(*

short summary
==================
This class tests all methods of REAL assertions
with various combinations of inputs and checks expected 
outputs are satisfied or not

.. <legal notes>

legal notes
=================
| SPDX-FileCopyrightText: © 2022 ekvip automation GmbH <info@ekvip.de>
| SPDX-License-Identifier: Apache-2.0
| For details check: Apache-2.0_

.. _Apache-2.0: https://www.apache.org/licenses/LICENSE-2.0

.. </legal notes>

methods and properties
======================

*)


FUNCTION_BLOCK RealAssertionTests EXTENDS AbstractAssertorTest
VAR
	(* not a number *)
	NAN							:REAL;
	(* infinity *)
	INF							:REAL;
	(* -infinity *)
	MINUS_INF					:REAL;
	(* -0.0 (MSB is set only) *)
	MINUS_ZERO					:REAL;
	(* minimum subnormal value (all fraction bits and MSB set only) *)
	MIN_SUBNORMAL				:REAL;
	(* maximum subnormal value (all fraction bits are set only) *)
	MAX_SUBNORMAL				:REAL;
	(* smallest positive subnormal value (LSB set only)*)
	SMALLEST_POSITIVE_SUBNORMAL	:REAL;
	(* smallest negative subnormal value (LSB and MSB set only)*)
	SMALLEST_NEGATIVE_SUBNORMAL	:REAL;
END_VAR
VAR CONSTANT
	(* prefix to unify the test names *)
	TEST_NAME_PREFIX					:STRING := 'assert.float.single.';
	(* max value of real *)
	MAX_NON_SPECIAL						:REAL := 3.402823E+38;
	(* min value of real *)
	MIN_NON_SPECIAL						:REAL := -3.402823E+38;
	(* 0.0 *)
	ZERO								:REAL := 0.0;
	(* 1% *)
	ONE_PERCENT							:REAL := 0.01;
	(* 1‰ *)
	ONE_PERMILLE						:REAL := 0.001;
	(* bit number of the sign bit *)
	SIGN								:USINT := 31;
	(* binary value of 0.0 *)
	BINARY_ZERO							:DWORD := 16#0000_0000;
	(* binary value of -0.0 *)
	BINARY_MINUS_ZERO					:DWORD := 16#8000_0000;
	(* binary value of inf *)
	BINARY_INFINITY						:DWORD := 16#7F80_0000;
	(* binary value of -inf *)
	BINARY_NEGATIVE_INFINITY			:DWORD := 16#FF80_0000;
	(* mask to filter the exponent of the number *)
	MASK_FOR_EXPONENT					:DWORD := 16#7F80_0000;
	(* minimum denormalized number *)
	BINARY_MIN_SUBNORMAL				:DWORD := 16#807F_FFFF;
	(* maximum denormalized number*)
	BINARY_MAX_SUBNORMAL				:DWORD := 16#007F_FFFF;
	(* smallest positive denormalizied number greater than zero *)
	BINARY_SMALLEST_POSITIVE_SUBNORMAL	:DWORD := 16#0000_0001;
	(* smallest negative denormalizied number greater than minus zero *)
	BINARY_SMALLEST_NEGATIVE_SUBNORMAL	:DWORD := 16#8000_0001;
	(* smallest positive signaling NaN *)
	BINARY_POSITIVE_SIGNALING_NAN		:DWORD := 16#7F80_0001;
END_VAR

THIS^.runValueIsEqualToTests();
THIS^.runValueIsGreaterThanTests();
THIS^.runValueIsInRangeOfTests();
THIS^.runValueIsLessThanTests();
THIS^.runValueIsMaxTests();
THIS^.runValueIsMinTests();
THIS^.runValueIsNotEqualToTests();
THIS^.runValueIsANumberTests();
THIS^.runValueIsFiniteTests();
THIS^.runValueIsInfiniteTests();
THIS^.runValueIsNaNTests();
THIS^.runValueIsNegativeTests();
THIS^.runValueIsPositiveTests();
THIS^.runValueIsNegativeInfiniteTests();
THIS^.runValueIsPositiveInfiniteTests();
THIS^.runValueIsNegativeZeroTests();
THIS^.runValueIsPositiveZeroTests();
THIS^.runValueIsNormalTests();
THIS^.runValueIsNotNegativeInfiniteTests();
THIS^.runValueIsNotPositiveInfiniteTests();
THIS^.runValueIsNotSpecialTests();
THIS^.runValueIsSpecialTests();
THIS^.runValueIsSubnormalTests();

(*

short summary
=============
It attaches the container with the class to test
and it sets the special numbers from `IEEE 754`_ standard

.. _IEEE 754: https://en.wikipedia.org/wiki/IEEE_754

legal notes
=================
| SPDX-FileCopyrightText: © 2023 ekvip automation GmbH <info@ekvip.de>
| SPDX-License-Identifier: Apache-2.0
| For details check: Apache-2.0_

.. _Apache-2.0: https://www.apache.org/licenses/LICENSE-2.0

.. </legal notes>

parameters
==========

*)

METHOD FB_init :BOOL
VAR_INPUT
	(* if TRUE, the retain variables are initialized (warm start / cold start) *)
    bInitRetains	:BOOL;
	(* if TRUE, the instance afterwards gets moved into the copy code (online change) *)
    bInCopyCode		:BOOL;
	(* container with the class to test *)
	classToBeTested :IAssertorContainer;
END_VAR
VAR
	{attribute 'hide'}
	newHashstate3		:CNM_AbstractObject.Hashcode;
	{attribute 'hide'}
	binaryNumberPointer	:POINTER TO DWORD;	
END_VAR
VAR CONSTANT
	{attribute 'hide'}
	NUMBER_OF_LEFT_SHIFTS		:UINT	:= 17;
	{attribute 'hide'}
	NUMBER_OF_LEFT_ROTATIONS	:UINT   := 45;
END_VAR
binaryNumberPointer := ADR(THIS^.NAN);
binaryNumberPointer^ := THIS^.BINARY_POSITIVE_SIGNALING_NAN;

binaryNumberPointer := ADR(THIS^.INF);
binaryNumberPointer^ := THIS^.BINARY_INFINITY;

binaryNumberPointer := ADR(THIS^.MINUS_INF);
binaryNumberPointer^ := THIS^.BINARY_NEGATIVE_INFINITY;

binaryNumberPointer := ADR(THIS^.MINUS_ZERO);
binaryNumberPointer^ := THIS^.BINARY_MINUS_ZERO;

binaryNumberPointer := ADR(THIS^.MIN_SUBNORMAL);
binaryNumberPointer^ := THIS^.BINARY_MIN_SUBNORMAL; 

binaryNumberPointer := ADR(THIS^.MAX_SUBNORMAL);
binaryNumberPointer^ := THIS^.BINARY_MAX_SUBNORMAL; 

binaryNumberPointer := ADR(THIS^.SMALLEST_POSITIVE_SUBNORMAL);
binaryNumberPointer^ := THIS^.BINARY_SMALLEST_POSITIVE_SUBNORMAL; 

binaryNumberPointer := ADR(THIS^.SMALLEST_NEGATIVE_SUBNORMAL);
binaryNumberPointer^ := THIS^.BINARY_SMALLEST_NEGATIVE_SUBNORMAL;
END_METHOD

(*

short summary
==================
This test method is a helper function to create a unified test name

.. <legal notes>

legal notes
=================
| SPDX-FileCopyrightText: © 2022 ekvip automation GmbH <info@ekvip.de>
| SPDX-License-Identifier: Apache-2.0
| For details check: Apache-2.0_

.. _Apache-2.0: https://www.apache.org/licenses/LICENSE-2.0

.. </legal notes>

parameters
==========

*)

METHOD PROTECTED getTestNameFor :Tc2_System.T_MaxString
VAR_INPUT
	(* name of the method to test, to create a unified test name *)
	nameOfMethodToTest	:Tc2_System.T_MaxString;
END_VAR
getTestNameFor := Tc2_Standard.CONCAT(THIS^.TEST_NAME_PREFIX, nameOfMethodToTest);
END_METHOD

(*

short summary
==================
This test method tests ``assert.float.single.valueIsANumber``
method of CNM_AssertionInterfaces library with various inputs

.. <legal notes>

legal notes
=================
| SPDX-FileCopyrightText: © 2022 ekvip automation GmbH <info@ekvip.de>
| SPDX-License-Identifier: Apache-2.0
| For details check: Apache-2.0_

.. _Apache-2.0: https://www.apache.org/licenses/LICENSE-2.0

.. </legal notes>

*)

METHOD runValueIsANumberTests
RETURN (NOT TcUnit.TEST_ORDERED(THIS^.getTestNameFor('valueIsANumber')));

THIS^.testValueIsANumber(THIS^.NAN);
THIS^.testValueIsANumber(THIS^.INF);
THIS^.testValueIsANumber(THIS^.MINUS_INF);
THIS^.testValueIsANumber(THIS^.MAX_NON_SPECIAL);
THIS^.testValueIsANumber(THIS^.MIN_NON_SPECIAL);
THIS^.testValueIsANumber(THIS^.ZERO);
THIS^.testValueIsANumber(THIS^.MINUS_ZERO);
THIS^.testValueIsANumber(THIS^.MAX_SUBNORMAL);
THIS^.testValueIsANumber(THIS^.MIN_SUBNORMAL);
THIS^.testValueIsANumber(THIS^.SMALLEST_NEGATIVE_SUBNORMAL);
THIS^.testValueIsANumber(THIS^.SMALLEST_POSITIVE_SUBNORMAL);
THIS^.testValueIsANumber(THIS^.ONE_PERCENT);
THIS^.testValueIsANumber(THIS^.ONE_PERMILLE);
THIS^.testValueIsANumber(THIS^.ONE_PERCENT * -1.0);
THIS^.testValueIsANumber(THIS^.ONE_PERMILLE * -1.0);

TcUnit.TEST_FINISHED();
END_METHOD

(*

short summary
==================
This test method tests ``assert.float.single.valueIsEqualTo``
method of CNM_AssertionInterfaces library with various inputs

.. <legal notes>

legal notes
=================
| SPDX-FileCopyrightText: © 2022 ekvip automation GmbH <info@ekvip.de>
| SPDX-License-Identifier: Apache-2.0
| For details check: Apache-2.0_

.. _Apache-2.0: https://www.apache.org/licenses/LICENSE-2.0

.. </legal notes>

*)

METHOD runValueIsEqualToTests
RETURN (NOT TcUnit.TEST_ORDERED(THIS^.getTestNameFor('valueIsEqualTo')));

THIS^.testValueIsEqualTo(
	valueToTest := THIS^.NAN,
	expected := THIS^.ONE_PERCENT,
	tolerance := THIS^.ONE_PERMILLE
);

THIS^.testValueIsEqualTo(
	valueToTest := THIS^.ONE_PERCENT,
	expected := THIS^.NAN,
	tolerance := THIS^.ONE_PERMILLE
);

THIS^.testValueIsEqualTo(
	valueToTest := THIS^.ONE_PERCENT,
	expected := THIS^.ONE_PERCENT,
	tolerance := THIS^.NAN
);

THIS^.testValueIsEqualTo(
	valueToTest := THIS^.NAN,
	expected := THIS^.NAN,
	tolerance := THIS^.ONE_PERCENT
);

THIS^.testValueIsEqualTo(
	valueToTest := THIS^.NAN,
	expected := THIS^.NAN,
	tolerance := THIS^.NAN
);

THIS^.testValueIsEqualTo(
	valueToTest := THIS^.INF,
	expected := THIS^.ONE_PERCENT,
	tolerance := THIS^.ONE_PERMILLE
);

THIS^.testValueIsEqualTo(
	valueToTest := THIS^.ONE_PERCENT,
	expected := THIS^.INF,
	tolerance := THIS^.ONE_PERMILLE
);

THIS^.testValueIsEqualTo(
	valueToTest := THIS^.ONE_PERCENT,
	expected := THIS^.ONE_PERCENT,
	tolerance := THIS^.INF
);

THIS^.testValueIsEqualTo(
	valueToTest := THIS^.INF,
	expected := THIS^.INF,
	tolerance := THIS^.ONE_PERCENT
);

THIS^.testValueIsEqualTo(
	valueToTest := THIS^.INF,
	expected := THIS^.INF,
	tolerance := THIS^.INF
);

THIS^.testValueIsEqualTo(
	valueToTest := THIS^.INF,
	expected := THIS^.MINUS_INF,
	tolerance := THIS^.INF
);

THIS^.testValueIsEqualTo(
	valueToTest := THIS^.MINUS_INF,
	expected := THIS^.ONE_PERCENT,
	tolerance := THIS^.ONE_PERMILLE
);

THIS^.testValueIsEqualTo(
	valueToTest := THIS^.ONE_PERCENT,
	expected := THIS^.MINUS_INF,
	tolerance := THIS^.ONE_PERMILLE
);

THIS^.testValueIsEqualTo(
	valueToTest := THIS^.ONE_PERCENT,
	expected := THIS^.ONE_PERCENT,
	tolerance := THIS^.MINUS_INF
);

THIS^.testValueIsEqualTo(
	valueToTest := THIS^.MINUS_INF,
	expected := THIS^.MINUS_INF,
	tolerance := THIS^.ONE_PERCENT
);

THIS^.testValueIsEqualTo(
	valueToTest := THIS^.MINUS_INF,
	expected := THIS^.MINUS_INF,
	tolerance := THIS^.MINUS_INF
);

THIS^.testValueIsEqualTo(
	valueToTest := THIS^.INF,
	expected := THIS^.MINUS_INF,
	tolerance := THIS^.INF
);

THIS^.testValueIsEqualTo(
	valueToTest := THIS^.MINUS_ZERO,
	expected := THIS^.SMALLEST_POSITIVE_SUBNORMAL,
	tolerance := THIS^.ONE_PERMILLE
);

THIS^.testValueIsEqualTo(
	valueToTest := THIS^.SMALLEST_POSITIVE_SUBNORMAL,
	expected := THIS^.MINUS_ZERO,
	tolerance := THIS^.ONE_PERMILLE
);

THIS^.testValueIsEqualTo(
	valueToTest := THIS^.SMALLEST_POSITIVE_SUBNORMAL,
	expected := THIS^.SMALLEST_POSITIVE_SUBNORMAL,
	tolerance := THIS^.MINUS_ZERO
);

THIS^.testValueIsEqualTo(
	valueToTest := THIS^.MINUS_ZERO,
	expected := THIS^.MINUS_ZERO,
	tolerance := THIS^.SMALLEST_POSITIVE_SUBNORMAL
);

THIS^.testValueIsEqualTo(
	valueToTest := THIS^.MINUS_ZERO,
	expected := THIS^.MINUS_ZERO,
	tolerance := THIS^.MINUS_ZERO
);

THIS^.testValueIsEqualTo(
	valueToTest := THIS^.MINUS_ZERO,
	expected := THIS^.ZERO,
	tolerance := THIS^.MINUS_ZERO
);

THIS^.testValueIsEqualTo(
	valueToTest := THIS^.ZERO,
	expected := THIS^.SMALLEST_POSITIVE_SUBNORMAL,
	tolerance := THIS^.ONE_PERMILLE
);

THIS^.testValueIsEqualTo(
	valueToTest := THIS^.SMALLEST_POSITIVE_SUBNORMAL,
	expected := THIS^.ZERO,
	tolerance := THIS^.ONE_PERMILLE
);

THIS^.testValueIsEqualTo(
	valueToTest := THIS^.SMALLEST_POSITIVE_SUBNORMAL,
	expected := THIS^.SMALLEST_POSITIVE_SUBNORMAL,
	tolerance := THIS^.ZERO
);

THIS^.testValueIsEqualTo(
	valueToTest := THIS^.ZERO,
	expected := THIS^.ZERO,
	tolerance := THIS^.SMALLEST_POSITIVE_SUBNORMAL
);

THIS^.testValueIsEqualTo(
	valueToTest := THIS^.ZERO,
	expected := THIS^.ZERO,
	tolerance := THIS^.ZERO
);

THIS^.testValueIsEqualTo(
	valueToTest := THIS^.ZERO,
	expected := THIS^.MINUS_ZERO,
	tolerance := THIS^.ZERO
);

THIS^.testValueIsEqualTo(
	valueToTest := THIS^.SMALLEST_POSITIVE_SUBNORMAL,
	expected := THIS^.ONE_PERCENT,
	tolerance := THIS^.ONE_PERMILLE
);

THIS^.testValueIsEqualTo(
	valueToTest := THIS^.ONE_PERCENT,
	expected := THIS^.SMALLEST_POSITIVE_SUBNORMAL,
	tolerance := THIS^.ONE_PERMILLE
);

THIS^.testValueIsEqualTo(
	valueToTest := THIS^.ONE_PERCENT,
	expected := THIS^.ONE_PERCENT,
	tolerance := THIS^.SMALLEST_POSITIVE_SUBNORMAL
);

THIS^.testValueIsEqualTo(
	valueToTest := THIS^.SMALLEST_POSITIVE_SUBNORMAL,
	expected := THIS^.SMALLEST_POSITIVE_SUBNORMAL,
	tolerance := THIS^.ONE_PERCENT
);

THIS^.testValueIsEqualTo(
	valueToTest := THIS^.SMALLEST_POSITIVE_SUBNORMAL,
	expected := THIS^.SMALLEST_POSITIVE_SUBNORMAL,
	tolerance := THIS^.SMALLEST_POSITIVE_SUBNORMAL
);

THIS^.testValueIsEqualTo(
	valueToTest := THIS^.SMALLEST_POSITIVE_SUBNORMAL,
	expected := THIS^.SMALLEST_NEGATIVE_SUBNORMAL,
	tolerance := THIS^.SMALLEST_POSITIVE_SUBNORMAL
);

THIS^.testValueIsEqualTo(
	valueToTest := THIS^.SMALLEST_NEGATIVE_SUBNORMAL,
	expected := THIS^.ONE_PERCENT,
	tolerance := THIS^.ONE_PERMILLE
);

THIS^.testValueIsEqualTo(
	valueToTest := THIS^.ONE_PERCENT,
	expected := THIS^.SMALLEST_NEGATIVE_SUBNORMAL,
	tolerance := THIS^.ONE_PERMILLE
);

THIS^.testValueIsEqualTo(
	valueToTest := THIS^.ONE_PERCENT,
	expected := THIS^.ONE_PERCENT,
	tolerance := THIS^.SMALLEST_NEGATIVE_SUBNORMAL
);

THIS^.testValueIsEqualTo(
	valueToTest := THIS^.SMALLEST_NEGATIVE_SUBNORMAL,
	expected := THIS^.SMALLEST_NEGATIVE_SUBNORMAL,
	tolerance := THIS^.ONE_PERCENT
);

THIS^.testValueIsEqualTo(
	valueToTest := THIS^.SMALLEST_NEGATIVE_SUBNORMAL,
	expected := THIS^.SMALLEST_NEGATIVE_SUBNORMAL,
	tolerance := THIS^.SMALLEST_NEGATIVE_SUBNORMAL
);

THIS^.testValueIsEqualTo(
	valueToTest := THIS^.SMALLEST_NEGATIVE_SUBNORMAL,
	expected := THIS^.SMALLEST_POSITIVE_SUBNORMAL,
	tolerance := THIS^.SMALLEST_NEGATIVE_SUBNORMAL
);

THIS^.testValueIsEqualTo(
	valueToTest := THIS^.MAX_SUBNORMAL,
	expected := THIS^.SMALLEST_POSITIVE_SUBNORMAL,
	tolerance := THIS^.SMALLEST_NEGATIVE_SUBNORMAL
);

THIS^.testValueIsEqualTo(
	valueToTest := THIS^.SMALLEST_POSITIVE_SUBNORMAL,
	expected := THIS^.MAX_SUBNORMAL,
	tolerance := THIS^.SMALLEST_NEGATIVE_SUBNORMAL
);

THIS^.testValueIsEqualTo(
	valueToTest := THIS^.SMALLEST_POSITIVE_SUBNORMAL,
	expected := THIS^.SMALLEST_POSITIVE_SUBNORMAL,
	tolerance := THIS^.MAX_SUBNORMAL
);

THIS^.testValueIsEqualTo(
	valueToTest := THIS^.MAX_SUBNORMAL,
	expected := THIS^.MAX_SUBNORMAL,
	tolerance := THIS^.SMALLEST_POSITIVE_SUBNORMAL
);

THIS^.testValueIsEqualTo(
	valueToTest := THIS^.MAX_SUBNORMAL,
	expected := THIS^.MAX_SUBNORMAL,
	tolerance := THIS^.MAX_SUBNORMAL
);

THIS^.testValueIsEqualTo(
	valueToTest := THIS^.MAX_SUBNORMAL,
	expected := THIS^.MIN_SUBNORMAL,
	tolerance := THIS^.MAX_SUBNORMAL
);
//
THIS^.testValueIsEqualTo(
	valueToTest := THIS^.MIN_SUBNORMAL,
	expected := THIS^.SMALLEST_POSITIVE_SUBNORMAL,
	tolerance := THIS^.SMALLEST_NEGATIVE_SUBNORMAL
);

THIS^.testValueIsEqualTo(
	valueToTest := THIS^.SMALLEST_POSITIVE_SUBNORMAL,
	expected := THIS^.MIN_SUBNORMAL,
	tolerance := THIS^.SMALLEST_NEGATIVE_SUBNORMAL
);

THIS^.testValueIsEqualTo(
	valueToTest := THIS^.SMALLEST_POSITIVE_SUBNORMAL,
	expected := THIS^.SMALLEST_POSITIVE_SUBNORMAL,
	tolerance := THIS^.MIN_SUBNORMAL
);

THIS^.testValueIsEqualTo(
	valueToTest := THIS^.MIN_SUBNORMAL,
	expected := THIS^.MIN_SUBNORMAL,
	tolerance := THIS^.SMALLEST_POSITIVE_SUBNORMAL
);

THIS^.testValueIsEqualTo(
	valueToTest := THIS^.MIN_SUBNORMAL,
	expected := THIS^.MIN_SUBNORMAL,
	tolerance := THIS^.MIN_SUBNORMAL
);

THIS^.testValueIsEqualTo(
	valueToTest := THIS^.MIN_SUBNORMAL,
	expected := THIS^.MAX_SUBNORMAL,
	tolerance := THIS^.MIN_SUBNORMAL
);

THIS^.testValueIsEqualTo(
	valueToTest := THIS^.MAX_NON_SPECIAL,
	expected := THIS^.SMALLEST_POSITIVE_SUBNORMAL,
	tolerance := THIS^.SMALLEST_NEGATIVE_SUBNORMAL
);

THIS^.testValueIsEqualTo(
	valueToTest := THIS^.SMALLEST_POSITIVE_SUBNORMAL,
	expected := THIS^.MAX_NON_SPECIAL,
	tolerance := THIS^.SMALLEST_NEGATIVE_SUBNORMAL
);

THIS^.testValueIsEqualTo(
	valueToTest := THIS^.SMALLEST_POSITIVE_SUBNORMAL,
	expected := THIS^.SMALLEST_POSITIVE_SUBNORMAL,
	tolerance := THIS^.MAX_NON_SPECIAL
);

THIS^.testValueIsEqualTo(
	valueToTest := THIS^.MAX_NON_SPECIAL,
	expected := THIS^.MAX_NON_SPECIAL,
	tolerance := THIS^.SMALLEST_POSITIVE_SUBNORMAL
);

THIS^.testValueIsEqualTo(
	valueToTest := THIS^.MAX_NON_SPECIAL,
	expected := THIS^.MAX_NON_SPECIAL,
	tolerance := THIS^.MAX_NON_SPECIAL
);

THIS^.testValueIsEqualTo(
	valueToTest := THIS^.MAX_NON_SPECIAL,
	expected := THIS^.MIN_NON_SPECIAL,
	tolerance := THIS^.MAX_NON_SPECIAL
);

THIS^.testValueIsEqualTo(
	valueToTest := THIS^.MIN_NON_SPECIAL,
	expected := THIS^.SMALLEST_POSITIVE_SUBNORMAL,
	tolerance := THIS^.SMALLEST_NEGATIVE_SUBNORMAL
);

THIS^.testValueIsEqualTo(
	valueToTest := THIS^.SMALLEST_POSITIVE_SUBNORMAL,
	expected := THIS^.MIN_NON_SPECIAL,
	tolerance := THIS^.SMALLEST_NEGATIVE_SUBNORMAL
);

THIS^.testValueIsEqualTo(
	valueToTest := THIS^.SMALLEST_POSITIVE_SUBNORMAL,
	expected := THIS^.SMALLEST_POSITIVE_SUBNORMAL,
	tolerance := THIS^.MIN_NON_SPECIAL
);

THIS^.testValueIsEqualTo(
	valueToTest := THIS^.MIN_NON_SPECIAL,
	expected := THIS^.MIN_NON_SPECIAL,
	tolerance := THIS^.SMALLEST_POSITIVE_SUBNORMAL
);

THIS^.testValueIsEqualTo(
	valueToTest := THIS^.MIN_NON_SPECIAL,
	expected := THIS^.MIN_NON_SPECIAL,
	tolerance := THIS^.MIN_NON_SPECIAL
);

THIS^.testValueIsEqualTo(
	valueToTest := THIS^.MAX_NON_SPECIAL,
	expected := THIS^.MIN_NON_SPECIAL,
	tolerance := THIS^.MAX_NON_SPECIAL
);

TcUnit.TEST_FINISHED();
END_METHOD

(*

short summary
==================
This test method tests ``assert.float.single.valueIsFinite``
method of CNM_AssertionInterfaces library with various inputs

.. <legal notes>

legal notes
=================
| SPDX-FileCopyrightText: © 2022 ekvip automation GmbH <info@ekvip.de>
| SPDX-License-Identifier: Apache-2.0
| For details check: Apache-2.0_

.. _Apache-2.0: https://www.apache.org/licenses/LICENSE-2.0

.. </legal notes>

*)

METHOD runValueIsFiniteTests
RETURN (NOT TcUnit.TEST_ORDERED(THIS^.getTestNameFor('valueIsFinite')));

THIS^.testValueIsFinite(THIS^.NAN);
THIS^.testValueIsFinite(THIS^.INF);
THIS^.testValueIsFinite(THIS^.MINUS_INF);
THIS^.testValueIsFinite(THIS^.MAX_NON_SPECIAL);
THIS^.testValueIsFinite(THIS^.MIN_NON_SPECIAL);
THIS^.testValueIsFinite(THIS^.ZERO);
THIS^.testValueIsFinite(THIS^.MINUS_ZERO);
THIS^.testValueIsFinite(THIS^.MAX_SUBNORMAL);
THIS^.testValueIsFinite(THIS^.MIN_SUBNORMAL);
THIS^.testValueIsFinite(THIS^.SMALLEST_NEGATIVE_SUBNORMAL);
THIS^.testValueIsFinite(THIS^.SMALLEST_POSITIVE_SUBNORMAL);
THIS^.testValueIsFinite(THIS^.ONE_PERCENT);
THIS^.testValueIsFinite(THIS^.ONE_PERMILLE);
THIS^.testValueIsFinite(THIS^.ONE_PERCENT * -1.0);
THIS^.testValueIsFinite(THIS^.ONE_PERMILLE * -1.0);

TcUnit.TEST_FINISHED();
END_METHOD

(*

short summary
==================
This test method tests ``assert.float.single.valueIsGreaterThan``
method of CNM_AssertionInterfaces library with various inputs

.. <legal notes>

legal notes
=================
| SPDX-FileCopyrightText: © 2022 ekvip automation GmbH <info@ekvip.de>
| SPDX-License-Identifier: Apache-2.0
| For details check: Apache-2.0_

.. _Apache-2.0: https://www.apache.org/licenses/LICENSE-2.0

.. </legal notes>

*)

METHOD runValueIsGreaterThanTests
RETURN (NOT TcUnit.TEST_ORDERED(THIS^.getTestNameFor('valueIsGreaterThan')));

THIS^.testValueIsGreaterThan(
	valueToTest := THIS^.NAN,
	lessValue := THIS^.NAN
);

THIS^.testValueIsGreaterThan(
	valueToTest := THIS^.ONE_PERCENT,
	lessValue := THIS^.NAN
);

THIS^.testValueIsGreaterThan(
	valueToTest := THIS^.NAN,
	lessValue := THIS^.ONE_PERCENT
);

THIS^.testValueIsGreaterThan(
	valueToTest := THIS^.INF,
	lessValue := THIS^.INF
);

THIS^.testValueIsGreaterThan(
	valueToTest := THIS^.MINUS_INF,
	lessValue := THIS^.MINUS_INF
);

THIS^.testValueIsGreaterThan(
	valueToTest := THIS^.MINUS_INF,
	lessValue := THIS^.INF
);

THIS^.testValueIsGreaterThan(
	valueToTest := THIS^.INF,
	lessValue := THIS^.MINUS_INF
);

THIS^.testValueIsGreaterThan(
	valueToTest := THIS^.ZERO,
	lessValue := THIS^.MINUS_ZERO
);

THIS^.testValueIsGreaterThan(
	valueToTest := THIS^.MINUS_ZERO,
	lessValue := THIS^.ZERO
);

THIS^.testValueIsGreaterThan(
	valueToTest := THIS^.MAX_SUBNORMAL,
	lessValue := THIS^.MIN_SUBNORMAL
);

THIS^.testValueIsGreaterThan(
	valueToTest := THIS^.MIN_SUBNORMAL,
	lessValue := THIS^.MAX_SUBNORMAL
);

THIS^.testValueIsGreaterThan(
	valueToTest := THIS^.MAX_SUBNORMAL,
	lessValue := THIS^.SMALLEST_NEGATIVE_SUBNORMAL
);

THIS^.testValueIsGreaterThan(
	valueToTest := THIS^.MIN_SUBNORMAL,
	lessValue := THIS^.SMALLEST_NEGATIVE_SUBNORMAL
);

THIS^.testValueIsGreaterThan(
	valueToTest := THIS^.MAX_SUBNORMAL,
	lessValue := THIS^.SMALLEST_POSITIVE_SUBNORMAL
);

THIS^.testValueIsGreaterThan(
	valueToTest := THIS^.MIN_SUBNORMAL,
	lessValue := THIS^.SMALLEST_POSITIVE_SUBNORMAL
);

THIS^.testValueIsGreaterThan(
	valueToTest := THIS^.SMALLEST_NEGATIVE_SUBNORMAL,
	lessValue := THIS^.SMALLEST_POSITIVE_SUBNORMAL
);

THIS^.testValueIsGreaterThan(
	valueToTest := THIS^.SMALLEST_POSITIVE_SUBNORMAL,
	lessValue := THIS^.SMALLEST_NEGATIVE_SUBNORMAL
);

THIS^.testValueIsGreaterThan(
	valueToTest := THIS^.ONE_PERCENT,
	lessValue := THIS^.ONE_PERMILLE
);

THIS^.testValueIsGreaterThan(
	valueToTest := THIS^.ONE_PERMILLE,
	lessValue := THIS^.ONE_PERCENT
);

THIS^.testValueIsGreaterThan(
	valueToTest := THIS^.ONE_PERMILLE,
	lessValue := THIS^.ONE_PERMILLE
);

THIS^.testValueIsGreaterThan(
	valueToTest := THIS^.ONE_PERCENT,
	lessValue := THIS^.ONE_PERCENT
);

THIS^.testValueIsGreaterThan(
	valueToTest := THIS^.MAX_NON_SPECIAL,
	lessValue := THIS^.MIN_NON_SPECIAL
);

THIS^.testValueIsGreaterThan(
	valueToTest := THIS^.MIN_NON_SPECIAL,
	lessValue := THIS^.MAX_NON_SPECIAL
);

THIS^.testValueIsGreaterThan(
	valueToTest := THIS^.MIN_NON_SPECIAL,
	lessValue := THIS^.MIN_NON_SPECIAL
);

THIS^.testValueIsGreaterThan(
	valueToTest := THIS^.MAX_NON_SPECIAL,
	lessValue := THIS^.MAX_NON_SPECIAL
);

TcUnit.TEST_FINISHED();
END_METHOD

(*

short summary
==================
This test method tests ``assert.float.single.valueIsInfinite``
method of CNM_AssertionInterfaces library with various inputs

.. <legal notes>

legal notes
=================
| SPDX-FileCopyrightText: © 2022 ekvip automation GmbH <info@ekvip.de>
| SPDX-License-Identifier: Apache-2.0
| For details check: Apache-2.0_

.. _Apache-2.0: https://www.apache.org/licenses/LICENSE-2.0

.. </legal notes>

*)

METHOD runValueIsInfiniteTests
RETURN (NOT TcUnit.TEST_ORDERED(THIS^.getTestNameFor('valueIsInfinite')));

THIS^.testValueIsInfinite(THIS^.NAN);
THIS^.testValueIsInfinite(THIS^.INF);
THIS^.testValueIsInfinite(THIS^.MINUS_INF);
THIS^.testValueIsInfinite(THIS^.MAX_NON_SPECIAL);
THIS^.testValueIsInfinite(THIS^.MIN_NON_SPECIAL);
THIS^.testValueIsInfinite(THIS^.ZERO);
THIS^.testValueIsInfinite(THIS^.MINUS_ZERO);
THIS^.testValueIsInfinite(THIS^.MAX_SUBNORMAL);
THIS^.testValueIsInfinite(THIS^.MIN_SUBNORMAL);
THIS^.testValueIsInfinite(THIS^.SMALLEST_NEGATIVE_SUBNORMAL);
THIS^.testValueIsInfinite(THIS^.SMALLEST_POSITIVE_SUBNORMAL);
THIS^.testValueIsInfinite(THIS^.ONE_PERCENT);
THIS^.testValueIsInfinite(THIS^.ONE_PERMILLE);
THIS^.testValueIsInfinite(THIS^.ONE_PERCENT * -1.0);
THIS^.testValueIsInfinite(THIS^.ONE_PERMILLE * -1.0);

TcUnit.TEST_FINISHED();
END_METHOD

(*

short summary
==================
This test method tests ``assert.dateAndTime.simple.dateOnly.valueIsInRangeOf``
method of CNM_AssertionInterfaces library with various inputs

.. <legal notes>

legal notes
=================
| SPDX-FileCopyrightText: © 2022 ekvip automation GmbH <info@ekvip.de>
| SPDX-License-Identifier: Apache-2.0
| For details check: Apache-2.0_

.. _Apache-2.0: https://www.apache.org/licenses/LICENSE-2.0

.. </legal notes>

*)

METHOD runValueIsInRangeOfTests
RETURN (NOT TcUnit.TEST_ORDERED(THIS^.getTestNameFor('valueIsInRangeOf')));

THIS^.testValueIsInRangeOf(
	lowerLimit := THIS^.NAN,
	valueToTest := THIS^.ONE_PERCENT,
	upperLimit := THIS^.ONE_PERMILLE
);

THIS^.testValueIsInRangeOf(
	lowerLimit := THIS^.ONE_PERCENT,
	valueToTest := THIS^.NAN,
	upperLimit := THIS^.ONE_PERMILLE
);

THIS^.testValueIsInRangeOf(
	lowerLimit := THIS^.ONE_PERCENT,
	valueToTest := THIS^.ONE_PERCENT,
	upperLimit := THIS^.NAN
);

THIS^.testValueIsInRangeOf(
	lowerLimit := THIS^.NAN,
	valueToTest := THIS^.NAN,
	upperLimit := THIS^.ONE_PERCENT
);

THIS^.testValueIsInRangeOf(
	lowerLimit := THIS^.NAN,
	valueToTest := THIS^.NAN,
	upperLimit := THIS^.NAN
);

THIS^.testValueIsInRangeOf(
	lowerLimit := THIS^.INF,
	valueToTest := THIS^.ONE_PERCENT,
	upperLimit := THIS^.ONE_PERMILLE
);

THIS^.testValueIsInRangeOf(
	lowerLimit := THIS^.ONE_PERCENT,
	valueToTest := THIS^.INF,
	upperLimit := THIS^.ONE_PERMILLE
);

THIS^.testValueIsInRangeOf(
	lowerLimit := THIS^.ONE_PERCENT,
	valueToTest := THIS^.ONE_PERCENT,
	upperLimit := THIS^.INF
);

THIS^.testValueIsInRangeOf(
	lowerLimit := THIS^.INF,
	valueToTest := THIS^.INF,
	upperLimit := THIS^.ONE_PERCENT
);

THIS^.testValueIsInRangeOf(
	lowerLimit := THIS^.INF,
	valueToTest := THIS^.INF,
	upperLimit := THIS^.INF
);

THIS^.testValueIsInRangeOf(
	lowerLimit := THIS^.INF,
	valueToTest := THIS^.MINUS_INF,
	upperLimit := THIS^.MINUS_INF
);

THIS^.testValueIsInRangeOf(
	lowerLimit := THIS^.MINUS_INF,
	valueToTest := THIS^.ONE_PERCENT,
	upperLimit := THIS^.ONE_PERMILLE
);

THIS^.testValueIsInRangeOf(
	lowerLimit := THIS^.ONE_PERCENT,
	valueToTest := THIS^.MINUS_INF,
	upperLimit := THIS^.ONE_PERMILLE
);

THIS^.testValueIsInRangeOf(
	lowerLimit := THIS^.ONE_PERCENT,
	valueToTest := THIS^.ONE_PERCENT,
	upperLimit := THIS^.MINUS_INF
);

THIS^.testValueIsInRangeOf(
	lowerLimit := THIS^.MINUS_INF,
	valueToTest := THIS^.MINUS_INF,
	upperLimit := THIS^.ONE_PERCENT
);

THIS^.testValueIsInRangeOf(
	lowerLimit := THIS^.MINUS_INF,
	valueToTest := THIS^.MINUS_INF,
	upperLimit := THIS^.MINUS_INF
);

THIS^.testValueIsInRangeOf(
	lowerLimit := THIS^.INF,
	valueToTest := THIS^.MINUS_INF,
	upperLimit := THIS^.INF
);

THIS^.testValueIsInRangeOf(
	lowerLimit := THIS^.MINUS_ZERO,
	valueToTest := THIS^.SMALLEST_POSITIVE_SUBNORMAL,
	upperLimit := THIS^.ONE_PERMILLE
);

THIS^.testValueIsInRangeOf(
	lowerLimit := THIS^.SMALLEST_POSITIVE_SUBNORMAL,
	valueToTest := THIS^.MINUS_ZERO,
	upperLimit := THIS^.ONE_PERMILLE
);

THIS^.testValueIsInRangeOf(
	lowerLimit := THIS^.SMALLEST_POSITIVE_SUBNORMAL,
	valueToTest := THIS^.SMALLEST_POSITIVE_SUBNORMAL,
	upperLimit := THIS^.MINUS_ZERO
);

THIS^.testValueIsInRangeOf(
	lowerLimit := THIS^.MINUS_ZERO,
	valueToTest := THIS^.MINUS_ZERO,
	upperLimit := THIS^.SMALLEST_POSITIVE_SUBNORMAL
);

THIS^.testValueIsInRangeOf(
	lowerLimit := THIS^.MINUS_ZERO,
	valueToTest := THIS^.MINUS_ZERO,
	upperLimit := THIS^.MINUS_ZERO
);

THIS^.testValueIsInRangeOf(
	lowerLimit := THIS^.MINUS_ZERO,
	valueToTest := THIS^.ZERO,
	upperLimit := THIS^.MINUS_ZERO
);

THIS^.testValueIsInRangeOf(
	lowerLimit := THIS^.ZERO,
	valueToTest := THIS^.SMALLEST_POSITIVE_SUBNORMAL,
	upperLimit := THIS^.ONE_PERMILLE
);

THIS^.testValueIsInRangeOf(
	lowerLimit := THIS^.SMALLEST_POSITIVE_SUBNORMAL,
	valueToTest := THIS^.ZERO,
	upperLimit := THIS^.ONE_PERMILLE
);

THIS^.testValueIsInRangeOf(
	lowerLimit := THIS^.SMALLEST_POSITIVE_SUBNORMAL,
	valueToTest := THIS^.SMALLEST_POSITIVE_SUBNORMAL,
	upperLimit := THIS^.ZERO
);

THIS^.testValueIsInRangeOf(
	lowerLimit := THIS^.ZERO,
	valueToTest := THIS^.ZERO,
	upperLimit := THIS^.SMALLEST_POSITIVE_SUBNORMAL
);

THIS^.testValueIsInRangeOf(
	lowerLimit := THIS^.ZERO,
	valueToTest := THIS^.ZERO,
	upperLimit := THIS^.ZERO
);

THIS^.testValueIsInRangeOf(
	lowerLimit := THIS^.ZERO,
	valueToTest := THIS^.MINUS_ZERO,
	upperLimit := THIS^.ZERO
);

THIS^.testValueIsInRangeOf(
	lowerLimit := THIS^.SMALLEST_POSITIVE_SUBNORMAL,
	valueToTest := THIS^.ONE_PERCENT,
	upperLimit := THIS^.ONE_PERMILLE
);

THIS^.testValueIsInRangeOf(
	lowerLimit := THIS^.ONE_PERCENT,
	valueToTest := THIS^.SMALLEST_POSITIVE_SUBNORMAL,
	upperLimit := THIS^.ONE_PERMILLE
);

THIS^.testValueIsInRangeOf(
	lowerLimit := THIS^.ONE_PERCENT,
	valueToTest := THIS^.ONE_PERCENT,
	upperLimit := THIS^.SMALLEST_POSITIVE_SUBNORMAL
);

THIS^.testValueIsInRangeOf(
	lowerLimit := THIS^.SMALLEST_POSITIVE_SUBNORMAL,
	valueToTest := THIS^.SMALLEST_POSITIVE_SUBNORMAL,
	upperLimit := THIS^.ONE_PERCENT
);

THIS^.testValueIsInRangeOf(
	lowerLimit := THIS^.SMALLEST_POSITIVE_SUBNORMAL,
	valueToTest := THIS^.SMALLEST_POSITIVE_SUBNORMAL,
	upperLimit := THIS^.SMALLEST_POSITIVE_SUBNORMAL
);

THIS^.testValueIsInRangeOf(
	lowerLimit := THIS^.SMALLEST_POSITIVE_SUBNORMAL,
	valueToTest := THIS^.SMALLEST_NEGATIVE_SUBNORMAL,
	upperLimit := THIS^.SMALLEST_NEGATIVE_SUBNORMAL
);

THIS^.testValueIsInRangeOf(
	lowerLimit := THIS^.SMALLEST_NEGATIVE_SUBNORMAL,
	valueToTest := THIS^.ONE_PERCENT,
	upperLimit := THIS^.ONE_PERMILLE
);

THIS^.testValueIsInRangeOf(
	lowerLimit := THIS^.ONE_PERCENT,
	valueToTest := THIS^.SMALLEST_NEGATIVE_SUBNORMAL,
	upperLimit := THIS^.ONE_PERMILLE
);

THIS^.testValueIsInRangeOf(
	lowerLimit := THIS^.ONE_PERCENT,
	valueToTest := THIS^.ONE_PERCENT,
	upperLimit := THIS^.SMALLEST_NEGATIVE_SUBNORMAL
);

THIS^.testValueIsInRangeOf(
	lowerLimit := THIS^.SMALLEST_NEGATIVE_SUBNORMAL,
	valueToTest := THIS^.SMALLEST_NEGATIVE_SUBNORMAL,
	upperLimit := THIS^.ONE_PERCENT
);

THIS^.testValueIsInRangeOf(
	lowerLimit := THIS^.SMALLEST_NEGATIVE_SUBNORMAL,
	valueToTest := THIS^.SMALLEST_NEGATIVE_SUBNORMAL,
	upperLimit := THIS^.SMALLEST_NEGATIVE_SUBNORMAL
);

THIS^.testValueIsInRangeOf(
	lowerLimit := THIS^.SMALLEST_NEGATIVE_SUBNORMAL,
	valueToTest := THIS^.SMALLEST_POSITIVE_SUBNORMAL,
	upperLimit := THIS^.SMALLEST_NEGATIVE_SUBNORMAL
);

THIS^.testValueIsInRangeOf(
	lowerLimit := THIS^.MAX_SUBNORMAL,
	valueToTest := THIS^.SMALLEST_POSITIVE_SUBNORMAL,
	upperLimit := THIS^.SMALLEST_NEGATIVE_SUBNORMAL
);

THIS^.testValueIsInRangeOf(
	lowerLimit := THIS^.SMALLEST_POSITIVE_SUBNORMAL,
	valueToTest := THIS^.MAX_SUBNORMAL,
	upperLimit := THIS^.SMALLEST_NEGATIVE_SUBNORMAL
);

THIS^.testValueIsInRangeOf(
	lowerLimit := THIS^.SMALLEST_POSITIVE_SUBNORMAL,
	valueToTest := THIS^.SMALLEST_POSITIVE_SUBNORMAL,
	upperLimit := THIS^.MAX_SUBNORMAL
);

THIS^.testValueIsInRangeOf(
	lowerLimit := THIS^.MAX_SUBNORMAL,
	valueToTest := THIS^.MAX_SUBNORMAL,
	upperLimit := THIS^.SMALLEST_POSITIVE_SUBNORMAL
);

THIS^.testValueIsInRangeOf(
	lowerLimit := THIS^.MAX_SUBNORMAL,
	valueToTest := THIS^.MAX_SUBNORMAL,
	upperLimit := THIS^.MAX_SUBNORMAL
);

THIS^.testValueIsInRangeOf(
	lowerLimit := THIS^.MAX_SUBNORMAL,
	valueToTest := THIS^.MIN_SUBNORMAL,
	upperLimit := THIS^.MAX_SUBNORMAL
);
//
THIS^.testValueIsInRangeOf(
	lowerLimit := THIS^.MIN_SUBNORMAL,
	valueToTest := THIS^.SMALLEST_POSITIVE_SUBNORMAL,
	upperLimit := THIS^.SMALLEST_NEGATIVE_SUBNORMAL
);

THIS^.testValueIsInRangeOf(
	lowerLimit := THIS^.SMALLEST_POSITIVE_SUBNORMAL,
	valueToTest := THIS^.MIN_SUBNORMAL,
	upperLimit := THIS^.SMALLEST_NEGATIVE_SUBNORMAL
);

THIS^.testValueIsInRangeOf(
	lowerLimit := THIS^.SMALLEST_POSITIVE_SUBNORMAL,
	valueToTest := THIS^.SMALLEST_POSITIVE_SUBNORMAL,
	upperLimit := THIS^.MIN_SUBNORMAL
);

THIS^.testValueIsInRangeOf(
	lowerLimit := THIS^.MIN_SUBNORMAL,
	valueToTest := THIS^.MIN_SUBNORMAL,
	upperLimit := THIS^.SMALLEST_POSITIVE_SUBNORMAL
);

THIS^.testValueIsInRangeOf(
	lowerLimit := THIS^.MIN_SUBNORMAL,
	valueToTest := THIS^.MIN_SUBNORMAL,
	upperLimit := THIS^.MIN_SUBNORMAL
);

THIS^.testValueIsInRangeOf(
	lowerLimit := THIS^.MIN_SUBNORMAL,
	valueToTest := THIS^.MAX_SUBNORMAL,
	upperLimit := THIS^.MIN_SUBNORMAL
);

THIS^.testValueIsInRangeOf(
	lowerLimit := THIS^.MAX_NON_SPECIAL,
	valueToTest := THIS^.SMALLEST_POSITIVE_SUBNORMAL,
	upperLimit := THIS^.SMALLEST_NEGATIVE_SUBNORMAL
);

THIS^.testValueIsInRangeOf(
	lowerLimit := THIS^.SMALLEST_POSITIVE_SUBNORMAL,
	valueToTest := THIS^.MAX_NON_SPECIAL,
	upperLimit := THIS^.SMALLEST_NEGATIVE_SUBNORMAL
);

THIS^.testValueIsInRangeOf(
	lowerLimit := THIS^.SMALLEST_POSITIVE_SUBNORMAL,
	valueToTest := THIS^.SMALLEST_POSITIVE_SUBNORMAL,
	upperLimit := THIS^.MAX_NON_SPECIAL
);

THIS^.testValueIsInRangeOf(
	lowerLimit := THIS^.MAX_NON_SPECIAL,
	valueToTest := THIS^.MAX_NON_SPECIAL,
	upperLimit := THIS^.SMALLEST_POSITIVE_SUBNORMAL
);

THIS^.testValueIsInRangeOf(
	lowerLimit := THIS^.MAX_NON_SPECIAL,
	valueToTest := THIS^.MAX_NON_SPECIAL,
	upperLimit := THIS^.MAX_NON_SPECIAL
);

THIS^.testValueIsInRangeOf(
	lowerLimit := THIS^.MAX_NON_SPECIAL,
	valueToTest := THIS^.MIN_NON_SPECIAL,
	upperLimit := THIS^.MAX_NON_SPECIAL
);

THIS^.testValueIsInRangeOf(
	lowerLimit := THIS^.MIN_NON_SPECIAL,
	valueToTest := THIS^.SMALLEST_POSITIVE_SUBNORMAL,
	upperLimit := THIS^.SMALLEST_NEGATIVE_SUBNORMAL
);

THIS^.testValueIsInRangeOf(
	lowerLimit := THIS^.SMALLEST_POSITIVE_SUBNORMAL,
	valueToTest := THIS^.MIN_NON_SPECIAL,
	upperLimit := THIS^.SMALLEST_NEGATIVE_SUBNORMAL
);

THIS^.testValueIsInRangeOf(
	lowerLimit := THIS^.SMALLEST_POSITIVE_SUBNORMAL,
	valueToTest := THIS^.SMALLEST_POSITIVE_SUBNORMAL,
	upperLimit := THIS^.MIN_NON_SPECIAL
);

THIS^.testValueIsInRangeOf(
	lowerLimit := THIS^.MIN_NON_SPECIAL,
	valueToTest := THIS^.MIN_NON_SPECIAL,
	upperLimit := THIS^.SMALLEST_POSITIVE_SUBNORMAL
);

THIS^.testValueIsInRangeOf(
	lowerLimit := THIS^.MIN_NON_SPECIAL,
	valueToTest := THIS^.MIN_NON_SPECIAL,
	upperLimit := THIS^.MIN_NON_SPECIAL
);

THIS^.testValueIsInRangeOf(
	lowerLimit := THIS^.MAX_NON_SPECIAL,
	valueToTest := THIS^.MIN_NON_SPECIAL,
	upperLimit := THIS^.MAX_NON_SPECIAL
);

TcUnit.TEST_FINISHED();
END_METHOD

(*

short summary
==================
This test method tests ``assert.float.single.valueIsLessThan``
method of CNM_AssertionInterfaces library with various inputs

.. <legal notes>

legal notes
=================
| SPDX-FileCopyrightText: © 2022 ekvip automation GmbH <info@ekvip.de>
| SPDX-License-Identifier: Apache-2.0
| For details check: Apache-2.0_

.. _Apache-2.0: https://www.apache.org/licenses/LICENSE-2.0

.. </legal notes>

*)

METHOD runValueIsLessThanTests
RETURN (NOT TcUnit.TEST_ORDERED(THIS^.getTestNameFor('valueIsLessThan')));

THIS^.testValueIsLessThan(
	valueToTest := THIS^.NAN,
	greaterValue := THIS^.NAN
);

THIS^.testValueIsLessThan(
	valueToTest := THIS^.ONE_PERCENT,
	greaterValue := THIS^.NAN
);

THIS^.testValueIsLessThan(
	valueToTest := THIS^.NAN,
	greaterValue := THIS^.ONE_PERCENT
);

THIS^.testValueIsLessThan(
	valueToTest := THIS^.INF,
	greaterValue := THIS^.INF
);

THIS^.testValueIsLessThan(
	valueToTest := THIS^.MINUS_INF,
	greaterValue := THIS^.MINUS_INF
);

THIS^.testValueIsLessThan(
	valueToTest := THIS^.MINUS_INF,
	greaterValue := THIS^.INF
);

THIS^.testValueIsLessThan(
	valueToTest := THIS^.INF,
	greaterValue := THIS^.MINUS_INF
);

THIS^.testValueIsLessThan(
	valueToTest := THIS^.ZERO,
	greaterValue := THIS^.MINUS_ZERO
);

THIS^.testValueIsLessThan(
	valueToTest := THIS^.MINUS_ZERO,
	greaterValue := THIS^.ZERO
);

THIS^.testValueIsLessThan(
	valueToTest := THIS^.MAX_SUBNORMAL,
	greaterValue := THIS^.MIN_SUBNORMAL
);

THIS^.testValueIsLessThan(
	valueToTest := THIS^.MIN_SUBNORMAL,
	greaterValue := THIS^.MAX_SUBNORMAL
);

THIS^.testValueIsLessThan(
	valueToTest := THIS^.MAX_SUBNORMAL,
	greaterValue := THIS^.SMALLEST_NEGATIVE_SUBNORMAL
);

THIS^.testValueIsLessThan(
	valueToTest := THIS^.MIN_SUBNORMAL,
	greaterValue := THIS^.SMALLEST_NEGATIVE_SUBNORMAL
);

THIS^.testValueIsLessThan(
	valueToTest := THIS^.MAX_SUBNORMAL,
	greaterValue := THIS^.SMALLEST_POSITIVE_SUBNORMAL
);

THIS^.testValueIsLessThan(
	valueToTest := THIS^.MIN_SUBNORMAL,
	greaterValue := THIS^.SMALLEST_POSITIVE_SUBNORMAL
);

THIS^.testValueIsLessThan(
	valueToTest := THIS^.SMALLEST_NEGATIVE_SUBNORMAL,
	greaterValue := THIS^.SMALLEST_POSITIVE_SUBNORMAL
);

THIS^.testValueIsLessThan(
	valueToTest := THIS^.SMALLEST_POSITIVE_SUBNORMAL,
	greaterValue := THIS^.SMALLEST_NEGATIVE_SUBNORMAL
);

THIS^.testValueIsLessThan(
	valueToTest := THIS^.ONE_PERCENT,
	greaterValue := THIS^.ONE_PERMILLE
);

THIS^.testValueIsLessThan(
	valueToTest := THIS^.ONE_PERMILLE,
	greaterValue := THIS^.ONE_PERCENT
);

THIS^.testValueIsLessThan(
	valueToTest := THIS^.ONE_PERMILLE,
	greaterValue := THIS^.ONE_PERMILLE
);

THIS^.testValueIsLessThan(
	valueToTest := THIS^.ONE_PERCENT,
	greaterValue := THIS^.ONE_PERCENT
);

THIS^.testValueIsLessThan(
	valueToTest := THIS^.MAX_NON_SPECIAL,
	greaterValue := THIS^.MIN_NON_SPECIAL
);

THIS^.testValueIsLessThan(
	valueToTest := THIS^.MIN_NON_SPECIAL,
	greaterValue := THIS^.MAX_NON_SPECIAL
);

THIS^.testValueIsLessThan(
	valueToTest := THIS^.MIN_NON_SPECIAL,
	greaterValue := THIS^.MIN_NON_SPECIAL
);

THIS^.testValueIsLessThan(
	valueToTest := THIS^.MAX_NON_SPECIAL,
	greaterValue := THIS^.MAX_NON_SPECIAL
);

TcUnit.TEST_FINISHED();
END_METHOD

(*

short summary
==================
This test method tests ``assert.float.single.valueIsMax``
method of CNM_AssertionInterfaces library with various inputs

.. <legal notes>

legal notes
=================
| SPDX-FileCopyrightText: © 2022 ekvip automation GmbH <info@ekvip.de>
| SPDX-License-Identifier: Apache-2.0
| For details check: Apache-2.0_

.. _Apache-2.0: https://www.apache.org/licenses/LICENSE-2.0

.. </legal notes>

*)

METHOD runValueIsMaxTests
RETURN (NOT TcUnit.TEST_ORDERED(THIS^.getTestNameFor('valueIsMax')));

THIS^.testValueIsMax(
	valueToTest := THIS^.NAN,
	maximumValue := THIS^.NAN
);

THIS^.testValueIsMax(
	valueToTest := THIS^.ONE_PERCENT,
	maximumValue := THIS^.NAN
);

THIS^.testValueIsMax(
	valueToTest := THIS^.NAN,
	maximumValue := THIS^.ONE_PERCENT
);

THIS^.testValueIsMax(
	valueToTest := THIS^.INF,
	maximumValue := THIS^.INF
);

THIS^.testValueIsMax(
	valueToTest := THIS^.MINUS_INF,
	maximumValue := THIS^.MINUS_INF
);

THIS^.testValueIsMax(
	valueToTest := THIS^.MINUS_INF,
	maximumValue := THIS^.INF
);

THIS^.testValueIsMax(
	valueToTest := THIS^.INF,
	maximumValue := THIS^.MINUS_INF
);

THIS^.testValueIsMax(
	valueToTest := THIS^.ZERO,
	maximumValue := THIS^.MINUS_ZERO
);

THIS^.testValueIsMax(
	valueToTest := THIS^.MINUS_ZERO,
	maximumValue := THIS^.ZERO
);

THIS^.testValueIsMax(
	valueToTest := THIS^.MAX_SUBNORMAL,
	maximumValue := THIS^.MIN_SUBNORMAL
);

THIS^.testValueIsMax(
	valueToTest := THIS^.MIN_SUBNORMAL,
	maximumValue := THIS^.MAX_SUBNORMAL
);

THIS^.testValueIsMax(
	valueToTest := THIS^.MAX_SUBNORMAL,
	maximumValue := THIS^.SMALLEST_NEGATIVE_SUBNORMAL
);

THIS^.testValueIsMax(
	valueToTest := THIS^.MIN_SUBNORMAL,
	maximumValue := THIS^.SMALLEST_NEGATIVE_SUBNORMAL
);

THIS^.testValueIsMax(
	valueToTest := THIS^.MAX_SUBNORMAL,
	maximumValue := THIS^.SMALLEST_POSITIVE_SUBNORMAL
);

THIS^.testValueIsMax(
	valueToTest := THIS^.MIN_SUBNORMAL,
	maximumValue := THIS^.SMALLEST_POSITIVE_SUBNORMAL
);

THIS^.testValueIsMax(
	valueToTest := THIS^.SMALLEST_NEGATIVE_SUBNORMAL,
	maximumValue := THIS^.SMALLEST_POSITIVE_SUBNORMAL
);

THIS^.testValueIsMax(
	valueToTest := THIS^.SMALLEST_POSITIVE_SUBNORMAL,
	maximumValue := THIS^.SMALLEST_NEGATIVE_SUBNORMAL
);

THIS^.testValueIsMax(
	valueToTest := THIS^.ONE_PERCENT,
	maximumValue := THIS^.ONE_PERMILLE
);

THIS^.testValueIsMax(
	valueToTest := THIS^.ONE_PERMILLE,
	maximumValue := THIS^.ONE_PERCENT
);

THIS^.testValueIsMax(
	valueToTest := THIS^.ONE_PERMILLE,
	maximumValue := THIS^.ONE_PERMILLE
);

THIS^.testValueIsMax(
	valueToTest := THIS^.ONE_PERCENT,
	maximumValue := THIS^.ONE_PERCENT
);

THIS^.testValueIsMax(
	valueToTest := THIS^.MAX_NON_SPECIAL,
	maximumValue := THIS^.MIN_NON_SPECIAL
);

THIS^.testValueIsMax(
	valueToTest := THIS^.MIN_NON_SPECIAL,
	maximumValue := THIS^.MAX_NON_SPECIAL
);

THIS^.testValueIsMax(
	valueToTest := THIS^.MIN_NON_SPECIAL,
	maximumValue := THIS^.MIN_NON_SPECIAL
);

THIS^.testValueIsMax(
	valueToTest := THIS^.MAX_NON_SPECIAL,
	maximumValue := THIS^.MAX_NON_SPECIAL
);

TcUnit.TEST_FINISHED();
END_METHOD

(*

short summary
==================
This test method tests ``assert.float.single.valueIsMin``
method of CNM_AssertionInterfaces library with various inputs

.. <legal notes>

legal notes
=================
| SPDX-FileCopyrightText: © 2022 ekvip automation GmbH <info@ekvip.de>
| SPDX-License-Identifier: Apache-2.0
| For details check: Apache-2.0_

.. _Apache-2.0: https://www.apache.org/licenses/LICENSE-2.0

.. </legal notes>

*)

METHOD runValueIsMinTests
RETURN (NOT TcUnit.TEST_ORDERED(THIS^.getTestNameFor('valueIsMin')));

THIS^.testValueIsMin(
	valueToTest := THIS^.NAN,
	minimumValue := THIS^.NAN
);

THIS^.testValueIsMin(
	valueToTest := THIS^.ONE_PERCENT,
	minimumValue := THIS^.NAN
);

THIS^.testValueIsMin(
	valueToTest := THIS^.NAN,
	minimumValue := THIS^.ONE_PERCENT
);

THIS^.testValueIsMin(
	valueToTest := THIS^.INF,
	minimumValue := THIS^.INF
);

THIS^.testValueIsMin(
	valueToTest := THIS^.MINUS_INF,
	minimumValue := THIS^.MINUS_INF
);

THIS^.testValueIsMin(
	valueToTest := THIS^.MINUS_INF,
	minimumValue := THIS^.INF
);

THIS^.testValueIsMin(
	valueToTest := THIS^.INF,
	minimumValue := THIS^.MINUS_INF
);

THIS^.testValueIsMin(
	valueToTest := THIS^.ZERO,
	minimumValue := THIS^.MINUS_ZERO
);

THIS^.testValueIsMin(
	valueToTest := THIS^.MINUS_ZERO,
	minimumValue := THIS^.ZERO
);

THIS^.testValueIsMin(
	valueToTest := THIS^.MAX_SUBNORMAL,
	minimumValue := THIS^.MIN_SUBNORMAL
);

THIS^.testValueIsMin(
	valueToTest := THIS^.MIN_SUBNORMAL,
	minimumValue := THIS^.MAX_SUBNORMAL
);

THIS^.testValueIsMin(
	valueToTest := THIS^.MAX_SUBNORMAL,
	minimumValue := THIS^.SMALLEST_NEGATIVE_SUBNORMAL
);

THIS^.testValueIsMin(
	valueToTest := THIS^.MIN_SUBNORMAL,
	minimumValue := THIS^.SMALLEST_NEGATIVE_SUBNORMAL
);

THIS^.testValueIsMin(
	valueToTest := THIS^.MAX_SUBNORMAL,
	minimumValue := THIS^.SMALLEST_POSITIVE_SUBNORMAL
);

THIS^.testValueIsMin(
	valueToTest := THIS^.MIN_SUBNORMAL,
	minimumValue := THIS^.SMALLEST_POSITIVE_SUBNORMAL
);

THIS^.testValueIsMin(
	valueToTest := THIS^.SMALLEST_NEGATIVE_SUBNORMAL,
	minimumValue := THIS^.SMALLEST_POSITIVE_SUBNORMAL
);

THIS^.testValueIsMin(
	valueToTest := THIS^.SMALLEST_POSITIVE_SUBNORMAL,
	minimumValue := THIS^.SMALLEST_NEGATIVE_SUBNORMAL
);

THIS^.testValueIsMin(
	valueToTest := THIS^.ONE_PERCENT,
	minimumValue := THIS^.ONE_PERMILLE
);

THIS^.testValueIsMin(
	valueToTest := THIS^.ONE_PERMILLE,
	minimumValue := THIS^.ONE_PERCENT
);

THIS^.testValueIsMin(
	valueToTest := THIS^.ONE_PERMILLE,
	minimumValue := THIS^.ONE_PERMILLE
);

THIS^.testValueIsMin(
	valueToTest := THIS^.ONE_PERCENT,
	minimumValue := THIS^.ONE_PERCENT
);

THIS^.testValueIsMin(
	valueToTest := THIS^.MAX_NON_SPECIAL,
	minimumValue := THIS^.MIN_NON_SPECIAL
);

THIS^.testValueIsMin(
	valueToTest := THIS^.MIN_NON_SPECIAL,
	minimumValue := THIS^.MAX_NON_SPECIAL
);

THIS^.testValueIsMin(
	valueToTest := THIS^.MIN_NON_SPECIAL,
	minimumValue := THIS^.MIN_NON_SPECIAL
);

THIS^.testValueIsMin(
	valueToTest := THIS^.MAX_NON_SPECIAL,
	minimumValue := THIS^.MAX_NON_SPECIAL
);

TcUnit.TEST_FINISHED();
END_METHOD

(*

short summary
==================
This test method tests ``assert.float.single.valueIsNaN``
method of CNM_AssertionInterfaces library with various inputs

.. <legal notes>

legal notes
=================
| SPDX-FileCopyrightText: © 2022 ekvip automation GmbH <info@ekvip.de>
| SPDX-License-Identifier: Apache-2.0
| For details check: Apache-2.0_

.. _Apache-2.0: https://www.apache.org/licenses/LICENSE-2.0

.. </legal notes>

*)

METHOD runValueIsNaNTests
RETURN (NOT TcUnit.TEST_ORDERED(THIS^.getTestNameFor('valueIsNaN')));

THIS^.testValueIsNaN(THIS^.NAN);
THIS^.testValueIsNaN(THIS^.INF);
THIS^.testValueIsNaN(THIS^.MINUS_INF);
THIS^.testValueIsNaN(THIS^.MAX_NON_SPECIAL);
THIS^.testValueIsNaN(THIS^.MIN_NON_SPECIAL);
THIS^.testValueIsNaN(THIS^.ZERO);
THIS^.testValueIsNaN(THIS^.MINUS_ZERO);
THIS^.testValueIsNaN(THIS^.MAX_SUBNORMAL);
THIS^.testValueIsNaN(THIS^.MIN_SUBNORMAL);
THIS^.testValueIsNaN(THIS^.SMALLEST_NEGATIVE_SUBNORMAL);
THIS^.testValueIsNaN(THIS^.SMALLEST_POSITIVE_SUBNORMAL);
THIS^.testValueIsNaN(THIS^.ONE_PERCENT);
THIS^.testValueIsNaN(THIS^.ONE_PERMILLE);
THIS^.testValueIsNaN(THIS^.ONE_PERCENT * -1.0);
THIS^.testValueIsNaN(THIS^.ONE_PERMILLE * -1.0);

TcUnit.TEST_FINISHED();
END_METHOD

(*

short summary
==================
This test method tests ``assert.float.single.valueIsNegativeInfinite``
method of CNM_AssertionInterfaces library with various inputs

.. <legal notes>

legal notes
=================
| SPDX-FileCopyrightText: © 2022 ekvip automation GmbH <info@ekvip.de>
| SPDX-License-Identifier: Apache-2.0
| For details check: Apache-2.0_

.. _Apache-2.0: https://www.apache.org/licenses/LICENSE-2.0

.. </legal notes>

*)

METHOD runValueIsNegativeInfiniteTests
RETURN (NOT TcUnit.TEST_ORDERED(THIS^.getTestNameFor('valueIsNegativeInfinite')));

THIS^.testValueIsNegativeInfinite(THIS^.NAN);
THIS^.testValueIsNegativeInfinite(THIS^.INF);
THIS^.testValueIsNegativeInfinite(THIS^.MINUS_INF);
THIS^.testValueIsNegativeInfinite(THIS^.MAX_NON_SPECIAL);
THIS^.testValueIsNegativeInfinite(THIS^.MIN_NON_SPECIAL);
THIS^.testValueIsNegativeInfinite(THIS^.ZERO);
THIS^.testValueIsNegativeInfinite(THIS^.MINUS_ZERO);
THIS^.testValueIsNegativeInfinite(THIS^.MAX_SUBNORMAL);
THIS^.testValueIsNegativeInfinite(THIS^.MIN_SUBNORMAL);
THIS^.testValueIsNegativeInfinite(THIS^.SMALLEST_NEGATIVE_SUBNORMAL);
THIS^.testValueIsNegativeInfinite(THIS^.SMALLEST_POSITIVE_SUBNORMAL);
THIS^.testValueIsNegativeInfinite(THIS^.ONE_PERCENT);
THIS^.testValueIsNegativeInfinite(THIS^.ONE_PERMILLE);
THIS^.testValueIsNegativeInfinite(THIS^.ONE_PERCENT * -1.0);
THIS^.testValueIsNegativeInfinite(THIS^.ONE_PERMILLE * -1.0);

TcUnit.TEST_FINISHED();
END_METHOD

(*

short summary
==================
This test method tests ``assert.float.single.valueIsNegative``
method of CNM_AssertionInterfaces library with various inputs

.. <legal notes>

legal notes
=================
| SPDX-FileCopyrightText: © 2022 ekvip automation GmbH <info@ekvip.de>
| SPDX-License-Identifier: Apache-2.0
| For details check: Apache-2.0_

.. _Apache-2.0: https://www.apache.org/licenses/LICENSE-2.0

.. </legal notes>

*)

METHOD runValueIsNegativeTests
RETURN (NOT TcUnit.TEST_ORDERED(THIS^.getTestNameFor('valueIsNegative')));

THIS^.testValueIsNegative(THIS^.NAN);
THIS^.testValueIsNegative(THIS^.INF);
THIS^.testValueIsNegative(THIS^.MINUS_INF);
THIS^.testValueIsNegative(THIS^.MAX_NON_SPECIAL);
THIS^.testValueIsNegative(THIS^.MIN_NON_SPECIAL);
THIS^.testValueIsNegative(THIS^.ZERO);
THIS^.testValueIsNegative(THIS^.MINUS_ZERO);
THIS^.testValueIsNegative(THIS^.MAX_SUBNORMAL);
THIS^.testValueIsNegative(THIS^.MIN_SUBNORMAL);
THIS^.testValueIsNegative(THIS^.SMALLEST_NEGATIVE_SUBNORMAL);
THIS^.testValueIsNegative(THIS^.SMALLEST_POSITIVE_SUBNORMAL);
THIS^.testValueIsNegative(THIS^.ONE_PERCENT);
THIS^.testValueIsNegative(THIS^.ONE_PERMILLE);
THIS^.testValueIsNegative(THIS^.ONE_PERCENT * -1.0);
THIS^.testValueIsNegative(THIS^.ONE_PERMILLE * -1.0);

TcUnit.TEST_FINISHED();
END_METHOD

(*

short summary
==================
This test method tests ``assert.float.single.valueIsNegativeZero``
method of CNM_AssertionInterfaces library with various inputs

.. <legal notes>

legal notes
=================
| SPDX-FileCopyrightText: © 2022 ekvip automation GmbH <info@ekvip.de>
| SPDX-License-Identifier: Apache-2.0
| For details check: Apache-2.0_

.. _Apache-2.0: https://www.apache.org/licenses/LICENSE-2.0

.. </legal notes>

*)

METHOD runValueIsNegativeZeroTests
RETURN (NOT TcUnit.TEST_ORDERED(THIS^.getTestNameFor('valueIsNegativeZero')));

THIS^.testValueIsNegativeZero(THIS^.NAN);
THIS^.testValueIsNegativeZero(THIS^.INF);
THIS^.testValueIsNegativeZero(THIS^.MINUS_INF);
THIS^.testValueIsNegativeZero(THIS^.MAX_NON_SPECIAL);
THIS^.testValueIsNegativeZero(THIS^.MIN_NON_SPECIAL);
THIS^.testValueIsNegativeZero(THIS^.ZERO);
THIS^.testValueIsNegativeZero(THIS^.MINUS_ZERO);
THIS^.testValueIsNegativeZero(THIS^.MAX_SUBNORMAL);
THIS^.testValueIsNegativeZero(THIS^.MIN_SUBNORMAL);
THIS^.testValueIsNegativeZero(THIS^.SMALLEST_NEGATIVE_SUBNORMAL);
THIS^.testValueIsNegativeZero(THIS^.SMALLEST_POSITIVE_SUBNORMAL);
THIS^.testValueIsNegativeZero(THIS^.ONE_PERCENT);
THIS^.testValueIsNegativeZero(THIS^.ONE_PERMILLE);
THIS^.testValueIsNegativeZero(THIS^.ONE_PERCENT * -1.0);
THIS^.testValueIsNegativeZero(THIS^.ONE_PERMILLE * -1.0);

TcUnit.TEST_FINISHED();
END_METHOD

(*

short summary
==================
This test method tests ``assert.float.single.valueIsNormal``
method of CNM_AssertionInterfaces library with various inputs

.. <legal notes>

legal notes
=================
| SPDX-FileCopyrightText: © 2022 ekvip automation GmbH <info@ekvip.de>
| SPDX-License-Identifier: Apache-2.0
| For details check: Apache-2.0_

.. _Apache-2.0: https://www.apache.org/licenses/LICENSE-2.0

.. </legal notes>

*)

METHOD runValueIsNormalTests
RETURN (NOT TcUnit.TEST_ORDERED(THIS^.getTestNameFor('valueIsNormal')));

THIS^.testValueIsNormal(THIS^.NAN);
THIS^.testValueIsNormal(THIS^.INF);
THIS^.testValueIsNormal(THIS^.MINUS_INF);
THIS^.testValueIsNormal(THIS^.MAX_NON_SPECIAL);
THIS^.testValueIsNormal(THIS^.MIN_NON_SPECIAL);
THIS^.testValueIsNormal(THIS^.ZERO);
THIS^.testValueIsNormal(THIS^.MINUS_ZERO);
THIS^.testValueIsNormal(THIS^.MAX_SUBNORMAL);
THIS^.testValueIsNormal(THIS^.MIN_SUBNORMAL);
THIS^.testValueIsNormal(THIS^.SMALLEST_NEGATIVE_SUBNORMAL);
THIS^.testValueIsNormal(THIS^.SMALLEST_POSITIVE_SUBNORMAL);
THIS^.testValueIsNormal(THIS^.ONE_PERCENT);
THIS^.testValueIsNormal(THIS^.ONE_PERMILLE);
THIS^.testValueIsNormal(THIS^.ONE_PERCENT * -1.0);
THIS^.testValueIsNormal(THIS^.ONE_PERMILLE * -1.0);

TcUnit.TEST_FINISHED();
END_METHOD

(*

short summary
==================
This test method tests ``assert.float.single.valueIsNotEqualTo``
method of CNM_AssertionInterfaces library with various inputs

.. <legal notes>

legal notes
=================
| SPDX-FileCopyrightText: © 2022 ekvip automation GmbH <info@ekvip.de>
| SPDX-License-Identifier: Apache-2.0
| For details check: Apache-2.0_

.. _Apache-2.0: https://www.apache.org/licenses/LICENSE-2.0

.. </legal notes>

*)

METHOD runValueIsNotEqualToTests
RETURN (NOT TcUnit.TEST_ORDERED(THIS^.getTestNameFor('valueIsNotEqualTo')));

THIS^.testValueIsNotEqualTo(
	valueToTest := THIS^.NAN,
	unexpectedValue := THIS^.ONE_PERCENT,
	tolerance := THIS^.ONE_PERMILLE
);

THIS^.testValueIsNotEqualTo(
	valueToTest := THIS^.ONE_PERCENT,
	unexpectedValue := THIS^.NAN,
	tolerance := THIS^.ONE_PERMILLE
);

THIS^.testValueIsNotEqualTo(
	valueToTest := THIS^.ONE_PERCENT,
	unexpectedValue := THIS^.ONE_PERCENT,
	tolerance := THIS^.NAN
);

THIS^.testValueIsNotEqualTo(
	valueToTest := THIS^.NAN,
	unexpectedValue := THIS^.NAN,
	tolerance := THIS^.ONE_PERCENT
);

THIS^.testValueIsNotEqualTo(
	valueToTest := THIS^.NAN,
	unexpectedValue := THIS^.NAN,
	tolerance := THIS^.NAN
);

THIS^.testValueIsNotEqualTo(
	valueToTest := THIS^.INF,
	unexpectedValue := THIS^.ONE_PERCENT,
	tolerance := THIS^.ONE_PERMILLE
);

THIS^.testValueIsNotEqualTo(
	valueToTest := THIS^.ONE_PERCENT,
	unexpectedValue := THIS^.INF,
	tolerance := THIS^.ONE_PERMILLE
);

THIS^.testValueIsNotEqualTo(
	valueToTest := THIS^.ONE_PERCENT,
	unexpectedValue := THIS^.ONE_PERCENT,
	tolerance := THIS^.INF
);

THIS^.testValueIsNotEqualTo(
	valueToTest := THIS^.INF,
	unexpectedValue := THIS^.INF,
	tolerance := THIS^.ONE_PERCENT
);

THIS^.testValueIsNotEqualTo(
	valueToTest := THIS^.INF,
	unexpectedValue := THIS^.INF,
	tolerance := THIS^.INF
);

THIS^.testValueIsNotEqualTo(
	valueToTest := THIS^.INF,
	unexpectedValue := THIS^.MINUS_INF,
	tolerance := THIS^.INF
);

THIS^.testValueIsNotEqualTo(
	valueToTest := THIS^.MINUS_INF,
	unexpectedValue := THIS^.ONE_PERCENT,
	tolerance := THIS^.ONE_PERMILLE
);

THIS^.testValueIsNotEqualTo(
	valueToTest := THIS^.ONE_PERCENT,
	unexpectedValue := THIS^.MINUS_INF,
	tolerance := THIS^.ONE_PERMILLE
);

THIS^.testValueIsNotEqualTo(
	valueToTest := THIS^.ONE_PERCENT,
	unexpectedValue := THIS^.ONE_PERCENT,
	tolerance := THIS^.MINUS_INF
);

THIS^.testValueIsNotEqualTo(
	valueToTest := THIS^.MINUS_INF,
	unexpectedValue := THIS^.MINUS_INF,
	tolerance := THIS^.ONE_PERCENT
);

THIS^.testValueIsNotEqualTo(
	valueToTest := THIS^.MINUS_INF,
	unexpectedValue := THIS^.MINUS_INF,
	tolerance := THIS^.MINUS_INF
);

THIS^.testValueIsNotEqualTo(
	valueToTest := THIS^.INF,
	unexpectedValue := THIS^.MINUS_INF,
	tolerance := THIS^.INF
);

THIS^.testValueIsNotEqualTo(
	valueToTest := THIS^.MINUS_ZERO,
	unexpectedValue := THIS^.SMALLEST_POSITIVE_SUBNORMAL,
	tolerance := THIS^.ONE_PERMILLE
);

THIS^.testValueIsNotEqualTo(
	valueToTest := THIS^.SMALLEST_POSITIVE_SUBNORMAL,
	unexpectedValue := THIS^.MINUS_ZERO,
	tolerance := THIS^.ONE_PERMILLE
);

THIS^.testValueIsNotEqualTo(
	valueToTest := THIS^.SMALLEST_POSITIVE_SUBNORMAL,
	unexpectedValue := THIS^.SMALLEST_POSITIVE_SUBNORMAL,
	tolerance := THIS^.MINUS_ZERO
);

THIS^.testValueIsNotEqualTo(
	valueToTest := THIS^.MINUS_ZERO,
	unexpectedValue := THIS^.MINUS_ZERO,
	tolerance := THIS^.SMALLEST_POSITIVE_SUBNORMAL
);

THIS^.testValueIsNotEqualTo(
	valueToTest := THIS^.MINUS_ZERO,
	unexpectedValue := THIS^.MINUS_ZERO,
	tolerance := THIS^.MINUS_ZERO
);

THIS^.testValueIsNotEqualTo(
	valueToTest := THIS^.MINUS_ZERO,
	unexpectedValue := THIS^.ZERO,
	tolerance := THIS^.MINUS_ZERO
);

THIS^.testValueIsNotEqualTo(
	valueToTest := THIS^.ZERO,
	unexpectedValue := THIS^.SMALLEST_POSITIVE_SUBNORMAL,
	tolerance := THIS^.ONE_PERMILLE
);

THIS^.testValueIsNotEqualTo(
	valueToTest := THIS^.SMALLEST_POSITIVE_SUBNORMAL,
	unexpectedValue := THIS^.ZERO,
	tolerance := THIS^.ONE_PERMILLE
);

THIS^.testValueIsNotEqualTo(
	valueToTest := THIS^.SMALLEST_POSITIVE_SUBNORMAL,
	unexpectedValue := THIS^.SMALLEST_POSITIVE_SUBNORMAL,
	tolerance := THIS^.ZERO
);

THIS^.testValueIsNotEqualTo(
	valueToTest := THIS^.ZERO,
	unexpectedValue := THIS^.ZERO,
	tolerance := THIS^.SMALLEST_POSITIVE_SUBNORMAL
);

THIS^.testValueIsNotEqualTo(
	valueToTest := THIS^.ZERO,
	unexpectedValue := THIS^.ZERO,
	tolerance := THIS^.ZERO
);

THIS^.testValueIsNotEqualTo(
	valueToTest := THIS^.ZERO,
	unexpectedValue := THIS^.MINUS_ZERO,
	tolerance := THIS^.ZERO
);

THIS^.testValueIsNotEqualTo(
	valueToTest := THIS^.SMALLEST_POSITIVE_SUBNORMAL,
	unexpectedValue := THIS^.ONE_PERCENT,
	tolerance := THIS^.ONE_PERMILLE
);

THIS^.testValueIsNotEqualTo(
	valueToTest := THIS^.ONE_PERCENT,
	unexpectedValue := THIS^.SMALLEST_POSITIVE_SUBNORMAL,
	tolerance := THIS^.ONE_PERMILLE
);

THIS^.testValueIsNotEqualTo(
	valueToTest := THIS^.ONE_PERCENT,
	unexpectedValue := THIS^.ONE_PERCENT,
	tolerance := THIS^.SMALLEST_POSITIVE_SUBNORMAL
);

THIS^.testValueIsNotEqualTo(
	valueToTest := THIS^.SMALLEST_POSITIVE_SUBNORMAL,
	unexpectedValue := THIS^.SMALLEST_POSITIVE_SUBNORMAL,
	tolerance := THIS^.ONE_PERCENT
);

THIS^.testValueIsNotEqualTo(
	valueToTest := THIS^.SMALLEST_POSITIVE_SUBNORMAL,
	unexpectedValue := THIS^.SMALLEST_POSITIVE_SUBNORMAL,
	tolerance := THIS^.SMALLEST_POSITIVE_SUBNORMAL
);

THIS^.testValueIsNotEqualTo(
	valueToTest := THIS^.SMALLEST_POSITIVE_SUBNORMAL,
	unexpectedValue := THIS^.SMALLEST_NEGATIVE_SUBNORMAL,
	tolerance := THIS^.SMALLEST_POSITIVE_SUBNORMAL
);

THIS^.testValueIsNotEqualTo(
	valueToTest := THIS^.SMALLEST_NEGATIVE_SUBNORMAL,
	unexpectedValue := THIS^.ONE_PERCENT,
	tolerance := THIS^.ONE_PERMILLE
);

THIS^.testValueIsNotEqualTo(
	valueToTest := THIS^.ONE_PERCENT,
	unexpectedValue := THIS^.SMALLEST_NEGATIVE_SUBNORMAL,
	tolerance := THIS^.ONE_PERMILLE
);

THIS^.testValueIsNotEqualTo(
	valueToTest := THIS^.ONE_PERCENT,
	unexpectedValue := THIS^.ONE_PERCENT,
	tolerance := THIS^.SMALLEST_NEGATIVE_SUBNORMAL
);

THIS^.testValueIsNotEqualTo(
	valueToTest := THIS^.SMALLEST_NEGATIVE_SUBNORMAL,
	unexpectedValue := THIS^.SMALLEST_NEGATIVE_SUBNORMAL,
	tolerance := THIS^.ONE_PERCENT
);

THIS^.testValueIsNotEqualTo(
	valueToTest := THIS^.SMALLEST_NEGATIVE_SUBNORMAL,
	unexpectedValue := THIS^.SMALLEST_NEGATIVE_SUBNORMAL,
	tolerance := THIS^.SMALLEST_NEGATIVE_SUBNORMAL
);

THIS^.testValueIsNotEqualTo(
	valueToTest := THIS^.SMALLEST_NEGATIVE_SUBNORMAL,
	unexpectedValue := THIS^.SMALLEST_POSITIVE_SUBNORMAL,
	tolerance := THIS^.SMALLEST_NEGATIVE_SUBNORMAL
);

THIS^.testValueIsNotEqualTo(
	valueToTest := THIS^.MAX_SUBNORMAL,
	unexpectedValue := THIS^.SMALLEST_POSITIVE_SUBNORMAL,
	tolerance := THIS^.SMALLEST_NEGATIVE_SUBNORMAL
);

THIS^.testValueIsNotEqualTo(
	valueToTest := THIS^.SMALLEST_POSITIVE_SUBNORMAL,
	unexpectedValue := THIS^.MAX_SUBNORMAL,
	tolerance := THIS^.SMALLEST_NEGATIVE_SUBNORMAL
);

THIS^.testValueIsNotEqualTo(
	valueToTest := THIS^.SMALLEST_POSITIVE_SUBNORMAL,
	unexpectedValue := THIS^.SMALLEST_POSITIVE_SUBNORMAL,
	tolerance := THIS^.MAX_SUBNORMAL
);

THIS^.testValueIsNotEqualTo(
	valueToTest := THIS^.MAX_SUBNORMAL,
	unexpectedValue := THIS^.MAX_SUBNORMAL,
	tolerance := THIS^.SMALLEST_POSITIVE_SUBNORMAL
);

THIS^.testValueIsNotEqualTo(
	valueToTest := THIS^.MAX_SUBNORMAL,
	unexpectedValue := THIS^.MAX_SUBNORMAL,
	tolerance := THIS^.MAX_SUBNORMAL
);

THIS^.testValueIsNotEqualTo(
	valueToTest := THIS^.MAX_SUBNORMAL,
	unexpectedValue := THIS^.MIN_SUBNORMAL,
	tolerance := THIS^.MAX_SUBNORMAL
);
//
THIS^.testValueIsNotEqualTo(
	valueToTest := THIS^.MIN_SUBNORMAL,
	unexpectedValue := THIS^.SMALLEST_POSITIVE_SUBNORMAL,
	tolerance := THIS^.SMALLEST_NEGATIVE_SUBNORMAL
);

THIS^.testValueIsNotEqualTo(
	valueToTest := THIS^.SMALLEST_POSITIVE_SUBNORMAL,
	unexpectedValue := THIS^.MIN_SUBNORMAL,
	tolerance := THIS^.SMALLEST_NEGATIVE_SUBNORMAL
);

THIS^.testValueIsNotEqualTo(
	valueToTest := THIS^.SMALLEST_POSITIVE_SUBNORMAL,
	unexpectedValue := THIS^.SMALLEST_POSITIVE_SUBNORMAL,
	tolerance := THIS^.MIN_SUBNORMAL
);

THIS^.testValueIsNotEqualTo(
	valueToTest := THIS^.MIN_SUBNORMAL,
	unexpectedValue := THIS^.MIN_SUBNORMAL,
	tolerance := THIS^.SMALLEST_POSITIVE_SUBNORMAL
);

THIS^.testValueIsNotEqualTo(
	valueToTest := THIS^.MIN_SUBNORMAL,
	unexpectedValue := THIS^.MIN_SUBNORMAL,
	tolerance := THIS^.MIN_SUBNORMAL
);

THIS^.testValueIsNotEqualTo(
	valueToTest := THIS^.MIN_SUBNORMAL,
	unexpectedValue := THIS^.MAX_SUBNORMAL,
	tolerance := THIS^.MIN_SUBNORMAL
);

THIS^.testValueIsNotEqualTo(
	valueToTest := THIS^.MAX_NON_SPECIAL,
	unexpectedValue := THIS^.SMALLEST_POSITIVE_SUBNORMAL,
	tolerance := THIS^.SMALLEST_NEGATIVE_SUBNORMAL
);

THIS^.testValueIsNotEqualTo(
	valueToTest := THIS^.SMALLEST_POSITIVE_SUBNORMAL,
	unexpectedValue := THIS^.MAX_NON_SPECIAL,
	tolerance := THIS^.SMALLEST_NEGATIVE_SUBNORMAL
);

THIS^.testValueIsNotEqualTo(
	valueToTest := THIS^.SMALLEST_POSITIVE_SUBNORMAL,
	unexpectedValue := THIS^.SMALLEST_POSITIVE_SUBNORMAL,
	tolerance := THIS^.MAX_NON_SPECIAL
);

THIS^.testValueIsNotEqualTo(
	valueToTest := THIS^.MAX_NON_SPECIAL,
	unexpectedValue := THIS^.MAX_NON_SPECIAL,
	tolerance := THIS^.SMALLEST_POSITIVE_SUBNORMAL
);

THIS^.testValueIsNotEqualTo(
	valueToTest := THIS^.MAX_NON_SPECIAL,
	unexpectedValue := THIS^.MAX_NON_SPECIAL,
	tolerance := THIS^.MAX_NON_SPECIAL
);

THIS^.testValueIsNotEqualTo(
	valueToTest := THIS^.MAX_NON_SPECIAL,
	unexpectedValue := THIS^.MIN_NON_SPECIAL,
	tolerance := THIS^.MAX_NON_SPECIAL
);

THIS^.testValueIsNotEqualTo(
	valueToTest := THIS^.MIN_NON_SPECIAL,
	unexpectedValue := THIS^.SMALLEST_POSITIVE_SUBNORMAL,
	tolerance := THIS^.SMALLEST_NEGATIVE_SUBNORMAL
);

THIS^.testValueIsNotEqualTo(
	valueToTest := THIS^.SMALLEST_POSITIVE_SUBNORMAL,
	unexpectedValue := THIS^.MIN_NON_SPECIAL,
	tolerance := THIS^.SMALLEST_NEGATIVE_SUBNORMAL
);

THIS^.testValueIsNotEqualTo(
	valueToTest := THIS^.SMALLEST_POSITIVE_SUBNORMAL,
	unexpectedValue := THIS^.SMALLEST_POSITIVE_SUBNORMAL,
	tolerance := THIS^.MIN_NON_SPECIAL
);

THIS^.testValueIsNotEqualTo(
	valueToTest := THIS^.MIN_NON_SPECIAL,
	unexpectedValue := THIS^.MIN_NON_SPECIAL,
	tolerance := THIS^.SMALLEST_POSITIVE_SUBNORMAL
);

THIS^.testValueIsNotEqualTo(
	valueToTest := THIS^.MIN_NON_SPECIAL,
	unexpectedValue := THIS^.MIN_NON_SPECIAL,
	tolerance := THIS^.MIN_NON_SPECIAL
);

THIS^.testValueIsNotEqualTo(
	valueToTest := THIS^.MAX_NON_SPECIAL,
	unexpectedValue := THIS^.MIN_NON_SPECIAL,
	tolerance := THIS^.MAX_NON_SPECIAL
);

TcUnit.TEST_FINISHED();
END_METHOD

(*

short summary
==================
This test method tests ``assert.float.single.valueIsNotNegativeInfinite``
method of CNM_AssertionInterfaces library with various inputs

.. <legal notes>

legal notes
=================
| SPDX-FileCopyrightText: © 2022 ekvip automation GmbH <info@ekvip.de>
| SPDX-License-Identifier: Apache-2.0
| For details check: Apache-2.0_

.. _Apache-2.0: https://www.apache.org/licenses/LICENSE-2.0

.. </legal notes>

*)

METHOD runValueIsNotNegativeInfiniteTests
RETURN (NOT TcUnit.TEST_ORDERED(THIS^.getTestNameFor('valueIsNotNegativeInfinite')));

THIS^.testValueIsNotNegativeInfinite(THIS^.NAN);
THIS^.testValueIsNotNegativeInfinite(THIS^.INF);
THIS^.testValueIsNotNegativeInfinite(THIS^.MINUS_INF);
THIS^.testValueIsNotNegativeInfinite(THIS^.MAX_NON_SPECIAL);
THIS^.testValueIsNotNegativeInfinite(THIS^.MIN_NON_SPECIAL);
THIS^.testValueIsNotNegativeInfinite(THIS^.ZERO);
THIS^.testValueIsNotNegativeInfinite(THIS^.MINUS_ZERO);
THIS^.testValueIsNotNegativeInfinite(THIS^.MAX_SUBNORMAL);
THIS^.testValueIsNotNegativeInfinite(THIS^.MIN_SUBNORMAL);
THIS^.testValueIsNotNegativeInfinite(THIS^.SMALLEST_NEGATIVE_SUBNORMAL);
THIS^.testValueIsNotNegativeInfinite(THIS^.SMALLEST_POSITIVE_SUBNORMAL);
THIS^.testValueIsNotNegativeInfinite(THIS^.ONE_PERCENT);
THIS^.testValueIsNotNegativeInfinite(THIS^.ONE_PERMILLE);
THIS^.testValueIsNotNegativeInfinite(THIS^.ONE_PERCENT * -1.0);
THIS^.testValueIsNotNegativeInfinite(THIS^.ONE_PERMILLE * -1.0);

TcUnit.TEST_FINISHED();
END_METHOD

(*

short summary
==================
This test method tests ``assert.float.single.valueIsNotPositiveInfinite``
method of CNM_AssertionInterfaces library with various inputs

.. <legal notes>

legal notes
=================
| SPDX-FileCopyrightText: © 2022 ekvip automation GmbH <info@ekvip.de>
| SPDX-License-Identifier: Apache-2.0
| For details check: Apache-2.0_

.. _Apache-2.0: https://www.apache.org/licenses/LICENSE-2.0

.. </legal notes>

*)

METHOD runValueIsNotPositiveInfiniteTests
RETURN (NOT TcUnit.TEST_ORDERED(THIS^.getTestNameFor('valueIsNotPositiveInfinite')));

THIS^.testValueIsNotPositiveInfinite(THIS^.NAN);
THIS^.testValueIsNotPositiveInfinite(THIS^.INF);
THIS^.testValueIsNotPositiveInfinite(THIS^.MINUS_INF);
THIS^.testValueIsNotPositiveInfinite(THIS^.MAX_NON_SPECIAL);
THIS^.testValueIsNotPositiveInfinite(THIS^.MIN_NON_SPECIAL);
THIS^.testValueIsNotPositiveInfinite(THIS^.ZERO);
THIS^.testValueIsNotPositiveInfinite(THIS^.MINUS_ZERO);
THIS^.testValueIsNotPositiveInfinite(THIS^.MAX_SUBNORMAL);
THIS^.testValueIsNotPositiveInfinite(THIS^.MIN_SUBNORMAL);
THIS^.testValueIsNotPositiveInfinite(THIS^.SMALLEST_NEGATIVE_SUBNORMAL);
THIS^.testValueIsNotPositiveInfinite(THIS^.SMALLEST_POSITIVE_SUBNORMAL);
THIS^.testValueIsNotPositiveInfinite(THIS^.ONE_PERCENT);
THIS^.testValueIsNotPositiveInfinite(THIS^.ONE_PERMILLE);
THIS^.testValueIsNotPositiveInfinite(THIS^.ONE_PERCENT * -1.0);
THIS^.testValueIsNotPositiveInfinite(THIS^.ONE_PERMILLE * -1.0);

TcUnit.TEST_FINISHED();
END_METHOD

(*

short summary
==================
This test method tests ``assert.float.single.valueIsNotSpecial``
method of CNM_AssertionInterfaces library with various inputs

.. <legal notes>

legal notes
=================
| SPDX-FileCopyrightText: © 2022 ekvip automation GmbH <info@ekvip.de>
| SPDX-License-Identifier: Apache-2.0
| For details check: Apache-2.0_

.. _Apache-2.0: https://www.apache.org/licenses/LICENSE-2.0

.. </legal notes>

*)

METHOD runValueIsNotSpecialTests
RETURN (NOT TcUnit.TEST_ORDERED(THIS^.getTestNameFor('valueIsNotSpecial')));

THIS^.testValueIsNotSpecial(THIS^.NAN);
THIS^.testValueIsNotSpecial(THIS^.INF);
THIS^.testValueIsNotSpecial(THIS^.MINUS_INF);
THIS^.testValueIsNotSpecial(THIS^.MAX_NON_SPECIAL);
THIS^.testValueIsNotSpecial(THIS^.MIN_NON_SPECIAL);
THIS^.testValueIsNotSpecial(THIS^.ZERO);
THIS^.testValueIsNotSpecial(THIS^.MINUS_ZERO);
THIS^.testValueIsNotSpecial(THIS^.MAX_SUBNORMAL);
THIS^.testValueIsNotSpecial(THIS^.MIN_SUBNORMAL);
THIS^.testValueIsNotSpecial(THIS^.SMALLEST_NEGATIVE_SUBNORMAL);
THIS^.testValueIsNotSpecial(THIS^.SMALLEST_POSITIVE_SUBNORMAL);
THIS^.testValueIsNotSpecial(THIS^.ONE_PERCENT);
THIS^.testValueIsNotSpecial(THIS^.ONE_PERMILLE);
THIS^.testValueIsNotSpecial(THIS^.ONE_PERCENT * -1.0);
THIS^.testValueIsNotSpecial(THIS^.ONE_PERMILLE * -1.0);

TcUnit.TEST_FINISHED();
END_METHOD

(*

short summary
==================
This test method tests ``assert.float.single.valueIsPositiveInfinite``
method of CNM_AssertionInterfaces library with various inputs

.. <legal notes>

legal notes
=================
| SPDX-FileCopyrightText: © 2022 ekvip automation GmbH <info@ekvip.de>
| SPDX-License-Identifier: Apache-2.0
| For details check: Apache-2.0_

.. _Apache-2.0: https://www.apache.org/licenses/LICENSE-2.0

.. </legal notes>

*)

METHOD runValueIsPositiveInfiniteTests
RETURN (NOT TcUnit.TEST_ORDERED(THIS^.getTestNameFor('valueIsPositiveInfinite')));

THIS^.testValueIsPositiveInfinite(THIS^.NAN);
THIS^.testValueIsPositiveInfinite(THIS^.INF);
THIS^.testValueIsPositiveInfinite(THIS^.MINUS_INF);
THIS^.testValueIsPositiveInfinite(THIS^.MAX_NON_SPECIAL);
THIS^.testValueIsPositiveInfinite(THIS^.MIN_NON_SPECIAL);
THIS^.testValueIsPositiveInfinite(THIS^.ZERO);
THIS^.testValueIsPositiveInfinite(THIS^.MINUS_ZERO);
THIS^.testValueIsPositiveInfinite(THIS^.MAX_SUBNORMAL);
THIS^.testValueIsPositiveInfinite(THIS^.MIN_SUBNORMAL);
THIS^.testValueIsPositiveInfinite(THIS^.SMALLEST_NEGATIVE_SUBNORMAL);
THIS^.testValueIsPositiveInfinite(THIS^.SMALLEST_POSITIVE_SUBNORMAL);
THIS^.testValueIsPositiveInfinite(THIS^.ONE_PERCENT);
THIS^.testValueIsPositiveInfinite(THIS^.ONE_PERMILLE);
THIS^.testValueIsPositiveInfinite(THIS^.ONE_PERCENT * -1.0);
THIS^.testValueIsPositiveInfinite(THIS^.ONE_PERMILLE * -1.0);

TcUnit.TEST_FINISHED();
END_METHOD

(*

short summary
==================
This test method tests ``assert.float.single.valueIsPositive``
method of CNM_AssertionInterfaces library with various inputs

.. <legal notes>

legal notes
=================
| SPDX-FileCopyrightText: © 2022 ekvip automation GmbH <info@ekvip.de>
| SPDX-License-Identifier: Apache-2.0
| For details check: Apache-2.0_

.. _Apache-2.0: https://www.apache.org/licenses/LICENSE-2.0

.. </legal notes>

*)

METHOD runValueIsPositiveTests
RETURN (NOT TcUnit.TEST_ORDERED(THIS^.getTestNameFor('valueIsPositive')));

THIS^.testValueIsPositive(THIS^.NAN);
THIS^.testValueIsPositive(THIS^.INF);
THIS^.testValueIsPositive(THIS^.MINUS_INF);
THIS^.testValueIsPositive(THIS^.MAX_NON_SPECIAL);
THIS^.testValueIsPositive(THIS^.MIN_NON_SPECIAL);
THIS^.testValueIsPositive(THIS^.ZERO);
THIS^.testValueIsPositive(THIS^.MINUS_ZERO);
THIS^.testValueIsPositive(THIS^.MAX_SUBNORMAL);
THIS^.testValueIsPositive(THIS^.MIN_SUBNORMAL);
THIS^.testValueIsPositive(THIS^.SMALLEST_NEGATIVE_SUBNORMAL);
THIS^.testValueIsPositive(THIS^.SMALLEST_POSITIVE_SUBNORMAL);
THIS^.testValueIsPositive(THIS^.ONE_PERCENT);
THIS^.testValueIsPositive(THIS^.ONE_PERMILLE);
THIS^.testValueIsPositive(THIS^.ONE_PERCENT * -1.0);
THIS^.testValueIsPositive(THIS^.ONE_PERMILLE * -1.0);

TcUnit.TEST_FINISHED();
END_METHOD

(*

short summary
==================
This test method tests ``assert.float.single.valueIsPositiveZero``
method of CNM_AssertionInterfaces library with various inputs

.. <legal notes>

legal notes
=================
| SPDX-FileCopyrightText: © 2022 ekvip automation GmbH <info@ekvip.de>
| SPDX-License-Identifier: Apache-2.0
| For details check: Apache-2.0_

.. _Apache-2.0: https://www.apache.org/licenses/LICENSE-2.0

.. </legal notes>

*)

METHOD runValueIsPositiveZeroTests
RETURN (NOT TcUnit.TEST_ORDERED(THIS^.getTestNameFor('valueIsPositiveZero')));

THIS^.testValueIsPositiveZero(THIS^.NAN);
THIS^.testValueIsPositiveZero(THIS^.INF);
THIS^.testValueIsPositiveZero(THIS^.MINUS_INF);
THIS^.testValueIsPositiveZero(THIS^.MAX_NON_SPECIAL);
THIS^.testValueIsPositiveZero(THIS^.MIN_NON_SPECIAL);
THIS^.testValueIsPositiveZero(THIS^.ZERO);
THIS^.testValueIsPositiveZero(THIS^.MINUS_ZERO);
THIS^.testValueIsPositiveZero(THIS^.MAX_SUBNORMAL);
THIS^.testValueIsPositiveZero(THIS^.MIN_SUBNORMAL);
THIS^.testValueIsPositiveZero(THIS^.SMALLEST_NEGATIVE_SUBNORMAL);
THIS^.testValueIsPositiveZero(THIS^.SMALLEST_POSITIVE_SUBNORMAL);
THIS^.testValueIsPositiveZero(THIS^.ONE_PERCENT);
THIS^.testValueIsPositiveZero(THIS^.ONE_PERMILLE);
THIS^.testValueIsPositiveZero(THIS^.ONE_PERCENT * -1.0);
THIS^.testValueIsPositiveZero(THIS^.ONE_PERMILLE * -1.0);

TcUnit.TEST_FINISHED();
END_METHOD

(*

short summary
==================
This test method tests ``assert.float.single.valueIsSpecial``
method of CNM_AssertionInterfaces library with various inputs

.. <legal notes>

legal notes
=================
| SPDX-FileCopyrightText: © 2022 ekvip automation GmbH <info@ekvip.de>
| SPDX-License-Identifier: Apache-2.0
| For details check: Apache-2.0_

.. _Apache-2.0: https://www.apache.org/licenses/LICENSE-2.0

.. </legal notes>

*)

METHOD runValueIsSpecialTests
RETURN (NOT TcUnit.TEST_ORDERED(THIS^.getTestNameFor('valueIsSpecial')));

THIS^.testValueIsSpecial(THIS^.NAN);
THIS^.testValueIsSpecial(THIS^.INF);
THIS^.testValueIsSpecial(THIS^.MINUS_INF);
THIS^.testValueIsSpecial(THIS^.MAX_NON_SPECIAL);
THIS^.testValueIsSpecial(THIS^.MIN_NON_SPECIAL);
THIS^.testValueIsSpecial(THIS^.ZERO);
THIS^.testValueIsSpecial(THIS^.MINUS_ZERO);
THIS^.testValueIsSpecial(THIS^.MAX_SUBNORMAL);
THIS^.testValueIsSpecial(THIS^.MIN_SUBNORMAL);
THIS^.testValueIsSpecial(THIS^.SMALLEST_NEGATIVE_SUBNORMAL);
THIS^.testValueIsSpecial(THIS^.SMALLEST_POSITIVE_SUBNORMAL);
THIS^.testValueIsSpecial(THIS^.ONE_PERCENT);
THIS^.testValueIsSpecial(THIS^.ONE_PERMILLE);
THIS^.testValueIsSpecial(THIS^.ONE_PERCENT * -1.0);
THIS^.testValueIsSpecial(THIS^.ONE_PERMILLE * -1.0);

TcUnit.TEST_FINISHED();
END_METHOD

(*

short summary
==================
This test method tests ``assert.float.single.valueIsSubnormal``
method of CNM_AssertionInterfaces library with various inputs

.. <legal notes>

legal notes
=================
| SPDX-FileCopyrightText: © 2022 ekvip automation GmbH <info@ekvip.de>
| SPDX-License-Identifier: Apache-2.0
| For details check: Apache-2.0_

.. _Apache-2.0: https://www.apache.org/licenses/LICENSE-2.0

.. </legal notes>

*)

METHOD runValueIsSubnormalTests
RETURN (NOT TcUnit.TEST_ORDERED(THIS^.getTestNameFor('valueIsSubnormal')));

THIS^.testValueIsSubnormal(THIS^.NAN);
THIS^.testValueIsSubnormal(THIS^.INF);
THIS^.testValueIsSubnormal(THIS^.MINUS_INF);
THIS^.testValueIsSubnormal(THIS^.MAX_NON_SPECIAL);
THIS^.testValueIsSubnormal(THIS^.MIN_NON_SPECIAL);
THIS^.testValueIsSubnormal(THIS^.ZERO);
THIS^.testValueIsSubnormal(THIS^.MINUS_ZERO);
THIS^.testValueIsSubnormal(THIS^.MAX_SUBNORMAL);
THIS^.testValueIsSubnormal(THIS^.MIN_SUBNORMAL);
THIS^.testValueIsSubnormal(THIS^.SMALLEST_NEGATIVE_SUBNORMAL);
THIS^.testValueIsSubnormal(THIS^.SMALLEST_POSITIVE_SUBNORMAL);
THIS^.testValueIsSubnormal(THIS^.ONE_PERCENT);
THIS^.testValueIsSubnormal(THIS^.ONE_PERMILLE);
THIS^.testValueIsSubnormal(THIS^.ONE_PERCENT * -1.0);
THIS^.testValueIsSubnormal(THIS^.ONE_PERMILLE * -1.0);

TcUnit.TEST_FINISHED();
END_METHOD

(*

short summary
==================
This test method tests ``assert.float.single.valueIsANumber``
method of CNM_AssertionInterfaces library, 
it provides the possibility to handover test data via parameter 

.. <legal notes>

legal notes
=================
| SPDX-FileCopyrightText: © 2022 ekvip automation GmbH <info@ekvip.de>
| SPDX-License-Identifier: Apache-2.0
| For details check: Apache-2.0_

.. _Apache-2.0: https://www.apache.org/licenses/LICENSE-2.0

.. </legal notes>

parameters
==========

*)

METHOD testValueIsANumber
VAR_INPUT
	(* for the test it's the parameter ``currentValue`` *)
	valueToTest	:REAL;	
END_VAR
VAR
	(* just the expectation if the assertion to test must be worng or true *)
	assertionIsWrong		:BOOL;
	(* contains the format string for the test message *)
	message					:Tc2_System.T_MaxString;
	(* TwinCAT printf with the test message *)
	messageStringBuilder	:Tc2_Utilities.FB_FormatString;
	(* value of the paramter ``valueToTest`` as string *)
	valueToTestAsString		:Tc2_System.T_MaxString;
END_VAR
THIS^.assertorContainer.resetAssertor();

assertionIsWrong := Tc2_Utilities.RealIsNaN(valueToTest);

message := SEL(
	assertionIsWrong,
	'currentValue is %s assertion must be TRUE', 
	'currentValue is %s assertion must be FALSE'
);

valueToTestAsString := TO_STRING(valueToTest);

messageStringBuilder(
	sFormat := message,
	arg1 := THIS^.AnyToArg(valueToTestAsString)
);

THIS^.assertorContainer.assertor.assert.float.single.valueIsANumber(
	currentValue := valueToTest,
	message := ''
);

THIS^.AssertEquals_BOOL(
	Expected 	:= assertionIsWrong,
	Actual 		:= THIS^.assertorContainer.wasAssertionWrong,
	Message 	:= messageStringBuilder.sOut
);
END_METHOD

(*

short summary
==================
This test method tests ``assert.float.single.valueIsEqualTo``
method of CNM_AssertionInterfaces library, 
it provides the possibility to handover test data via parameter 


.. <legal notes>

legal notes
=================
| SPDX-FileCopyrightText: © 2022 ekvip automation GmbH <info@ekvip.de>
| SPDX-License-Identifier: Apache-2.0
| For details check: Apache-2.0_

.. _Apache-2.0: https://www.apache.org/licenses/LICENSE-2.0

.. </legal notes>

parameters
==========

*)

METHOD testValueIsEqualTo 
VAR_INPUT
	(* for the test it's the parameter ``currentValue`` *)
	valueToTest	:REAL;
	(* for the test it's the parameter ``expectedValue`` *)
	expected	:REAL;
	(* for the test it's the parameter ``tolerance`` *)
	tolerance	:REAL;
END_VAR
VAR
	(* just the expectation if the assertion to test must be worng or true *)
	assertionIsWrong		:BOOL;
	(* contains the format string for the test message *)
	message					:Tc2_System.T_MaxString;
	(* TwinCAT printf with the test message *)
	messageStringBuilder	:Tc2_Utilities.FB_FormatString;
	(* just to cast *)
	binaryCurrentValue		:POINTER TO DWORD;
	(* just to cast *)
	binaryExpectedValue		:POINTER TO DWORD;
	(* value of the paramter ``valueToTest`` as string *)
	valueToTestAsString		:Tc2_System.T_MaxString;
	(* value of the paramter ``expected`` as string *)
	expectedAsString		:Tc2_System.T_MaxString;
	(* value of the paramter ``tolerance`` as string *)
	toleranceAsString		:Tc2_System.T_MaxString;	
END_VAR
THIS^.assertorContainer.resetAssertor();
IF (
	Tc2_Utilities.RealIsNaN(valueToTest)
	OR Tc2_Utilities.RealIsNaN(expected)
	OR Tc2_Utilities.RealIsNaN(tolerance)
) THEN
	assertionIsWrong := TRUE;
ELSIF (NOT Tc2_Utilities.RealIsFinite(tolerance)) THEN
	assertionIsWrong := FALSE;
ELSIF (Tc2_Utilities.RealIsFinite(valueToTest) <> Tc2_Utilities.RealIsFinite(expected)) THEN
	assertionIsWrong := TRUE; 
ELSIF (
	(NOT Tc2_Utilities.RealIsFinite(valueToTest))
	OR (NOT Tc2_Utilities.RealIsFinite(expected))
) THEN
	binaryCurrentValue := ADR(valueToTest);
	binaryExpectedValue := ADR(expected);
	assertionIsWrong := (binaryCurrentValue^.SIGN <> binaryExpectedValue^.SIGN);
ELSE
	assertionIsWrong := (
		((expected + ABS(tolerance)) < valueToTest)
		OR ((expected - ABS(tolerance)) > valueToTest)
	);
END_IF

message := SEL(
	assertionIsWrong,
	'currentValue is %s expectedValue is %s tolerance is %s assertion must be TRUE', 
	'currentValue is %s expectedValue is %s tolerance is %s assertion must be FALSE'
);

valueToTestAsString := TO_STRING(valueToTest);
expectedAsString := TO_STRING(expected);
toleranceAsString := TO_STRING(tolerance);

messageStringBuilder(
	sFormat := message,
	arg1 := THIS^.AnyToArg(valueToTestAsString),
	arg2 := THIS^.AnyToArg(expectedAsString),
	arg3 := THIS^.AnyToArg(toleranceAsString)
);

THIS^.assertorContainer.assertor.assert.float.single.valueIsEqualTo(
	currentValue	:= valueToTest,
	expectedValue	:= expected,
	tolerance       := tolerance,
	message			:= ''
);

THIS^.AssertEquals_BOOL(
	Expected 	:= assertionIsWrong,
	Actual 		:= THIS^.assertorContainer.wasAssertionWrong,
	Message 	:= messageStringBuilder.sOut
);
END_METHOD

(*

short summary
==================
This test method tests ``assert.float.single.valueIsFinite``
method of CNM_AssertionInterfaces library, 
it provides the possibility to handover test data via parameter 

.. <legal notes>

legal notes
=================
| SPDX-FileCopyrightText: © 2022 ekvip automation GmbH <info@ekvip.de>
| SPDX-License-Identifier: Apache-2.0
| For details check: Apache-2.0_

.. _Apache-2.0: https://www.apache.org/licenses/LICENSE-2.0

.. </legal notes>

parameters
==========

*)

METHOD testValueIsFinite
VAR_INPUT
	(* for the test it's the parameter ``currentValue`` *)
	valueToTest	:REAL;	
END_VAR
VAR
	(* just the expectation if the assertion to test must be worng or true *)
	assertionIsWrong		:BOOL;
	(* contains the format string for the test message *)
	message					:Tc2_System.T_MaxString;
	(* TwinCAT printf with the test message *)
	messageStringBuilder	:Tc2_Utilities.FB_FormatString;
	(* value of the paramter ``valueToTest`` as string *)
	valueToTestAsString		:Tc2_System.T_MaxString;
	(* binary value of the parameter ``valueToTest`` *)
	binaryValueToTest		:POINTER TO DWORD;
END_VAR
THIS^.assertorContainer.resetAssertor();

binaryValueToTest := ADR(valueToTest);
assertionIsWrong := (
	(binaryValueToTest^ = THIS^.BINARY_INFINITY)
	OR_ELSE (binaryValueToTest^ = THIS^.BINARY_NEGATIVE_INFINITY)
);

message := SEL(
	assertionIsWrong,
	'currentValue is %s assertion must be TRUE', 
	'currentValue is %s assertion must be FALSE'
);

valueToTestAsString := TO_STRING(valueToTest);

messageStringBuilder(
	sFormat := message,
	arg1 := THIS^.AnyToArg(valueToTestAsString)
);

THIS^.assertorContainer.assertor.assert.float.single.valueIsFinite(
	currentValue := valueToTest,
	message := ''
);

THIS^.AssertEquals_BOOL(
	Expected 	:= assertionIsWrong,
	Actual 		:= THIS^.assertorContainer.wasAssertionWrong,
	Message 	:= messageStringBuilder.sOut
);
END_METHOD

(*

short summary
==================
This test method tests ``assert.float.single.valueIsGreaterThan``
method of CNM_AssertionInterfaces library, 
it provides the possibility to handover test data via parameter 


.. <legal notes>

legal notes
=================
| SPDX-FileCopyrightText: © 2022 ekvip automation GmbH <info@ekvip.de>
| SPDX-License-Identifier: Apache-2.0
| For details check: Apache-2.0_

.. _Apache-2.0: https://www.apache.org/licenses/LICENSE-2.0

.. </legal notes>

parameters
==========

*)

METHOD testValueIsGreaterThan 
VAR_INPUT
	(* for the test it's the parameter ``currentValue`` *)
	valueToTest	:REAL;
	(* for the test it's the parameter ``lessValue`` *)
	lessValue	:REAL;
END_VAR
VAR
	(* just the expectation if the assertion to test must be worng or true *)
	assertionIsWrong		:BOOL;
	(* contains the format string for the test message *)
	message					:Tc2_System.T_MaxString;
	(* TwinCAT printf with the test message *)
	messageStringBuilder	:Tc2_Utilities.FB_FormatString;
	(* just to cast *)
	binaryCurrentValue		:POINTER TO DWORD;
	(* just to cast *)
	binaryLessValue			:POINTER TO DWORD;
	(* value of the paramter ``valueToTest`` as string *)
	valueToTestAsString		:Tc2_System.T_MaxString;
	(* value of the paramter ``lessValue`` as string *)
	lessValueAsString		:Tc2_System.T_MaxString;	
END_VAR
THIS^.assertorContainer.resetAssertor();

IF (Tc2_Utilities.RealIsNaN(valueToTest) OR Tc2_Utilities.RealIsNaN(lessValue)) THEN
	assertionIsWrong := TRUE;
ELSIF ((NOT Tc2_Utilities.RealIsFinite(valueToTest)) AND (NOT Tc2_Utilities.RealIsFinite(lessValue))) THEN
	binaryCurrentValue := ADR(valueToTest);
	binaryLessValue := ADR(lessValue);
	assertionIsWrong := (
		(binaryCurrentValue^.SIGN) //-inf
		OR (NOT binaryLessValue^.SIGN) //inf
	);
ELSIF ((NOT Tc2_Utilities.RealIsFinite(valueToTest)) AND (Tc2_Utilities.RealIsFinite(lessValue))) THEN
	binaryCurrentValue := ADR(valueToTest);
	assertionIsWrong := (binaryCurrentValue^.SIGN);
ELSIF (
	(Tc2_Utilities.RealIsFinite(valueToTest))
	AND (NOT Tc2_Utilities.RealIsFinite(lessValue))
) THEN
	binaryLessValue := ADR(lessValue);
	assertionIsWrong := (NOT binaryLessValue^.SIGN);
ELSE
	assertionIsWrong := (valueToTest <= lessValue);
END_IF

message := SEL(
	assertionIsWrong,
	'currentValue is %s lessValue is %s assertion must be TRUE', 
	'currentValue is %s lessValue is %s assertion must be FALSE'
);

valueToTestAsString := TO_STRING(valueToTest);
lessValueAsString := TO_STRING(lessValue);

messageStringBuilder(
	sFormat := message,
	arg1 := THIS^.AnyToArg(valueToTestAsString),
	arg2 := THIS^.AnyToArg(lessValueAsString)
);

THIS^.assertorContainer.assertor.assert.float.single.valueIsGreaterThan(
	currentValue	:= valueToTest,
	lessValue		:= lessValue,
	message			:= ''
);

THIS^.AssertEquals_BOOL(
	Expected 	:= assertionIsWrong,
	Actual 		:= THIS^.assertorContainer.wasAssertionWrong,
	Message 	:= messageStringBuilder.sOut
);
END_METHOD

(*

short summary
==================
This test method tests ``assert.float.single.valueIsInfinite``
method of CNM_AssertionInterfaces library, 
it provides the possibility to handover test data via parameter 

.. <legal notes>

legal notes
=================
| SPDX-FileCopyrightText: © 2022 ekvip automation GmbH <info@ekvip.de>
| SPDX-License-Identifier: Apache-2.0
| For details check: Apache-2.0_

.. _Apache-2.0: https://www.apache.org/licenses/LICENSE-2.0

.. </legal notes>

parameters
==========

*)

METHOD testValueIsInfinite
VAR_INPUT
	(* for the test it's the parameter ``currentValue`` *)
	valueToTest	:REAL;	
END_VAR
VAR
	(* just the expectation if the assertion to test must be worng or true *)
	assertionIsWrong		:BOOL;
	(* contains the format string for the test message *)
	message					:Tc2_System.T_MaxString;
	(* TwinCAT printf with the test message *)
	messageStringBuilder	:Tc2_Utilities.FB_FormatString;
	(* value of the paramter ``valueToTest`` as string *)
	valueToTestAsString		:Tc2_System.T_MaxString;
	(* binary value of the parameter ``valueToTest`` *)
	binaryValueToTest		:POINTER TO DWORD;
END_VAR
THIS^.assertorContainer.resetAssertor();

binaryValueToTest := ADR(valueToTest);
assertionIsWrong := (
	(binaryValueToTest^ <> THIS^.BINARY_INFINITY)
	AND_THEN (binaryValueToTest^ <> THIS^.BINARY_NEGATIVE_INFINITY)
);

message := SEL(
	assertionIsWrong,
	'currentValue is %s assertion must be TRUE', 
	'currentValue is %s assertion must be FALSE'
);

valueToTestAsString := TO_STRING(valueToTest);

messageStringBuilder(
	sFormat := message,
	arg1 := THIS^.AnyToArg(valueToTestAsString)
);

THIS^.assertorContainer.assertor.assert.float.single.valueIsInfinite(
	currentValue := valueToTest,
	message := ''
);

THIS^.AssertEquals_BOOL(
	Expected 	:= assertionIsWrong,
	Actual 		:= THIS^.assertorContainer.wasAssertionWrong,
	Message 	:= messageStringBuilder.sOut
);
END_METHOD

(*

short summary
==================
This test method tests ``assert.float.single.valueIsInRangeOf``
method of CNM_AssertionInterfaces library, 
it provides the possibility to handover test data via parameter 


.. <legal notes>

legal notes
=================
| SPDX-FileCopyrightText: © 2022 ekvip automation GmbH <info@ekvip.de>
| SPDX-License-Identifier: Apache-2.0
| For details check: Apache-2.0_

.. _Apache-2.0: https://www.apache.org/licenses/LICENSE-2.0

.. </legal notes>

parameters
==========

*)

METHOD testValueIsInRangeOf 
VAR_INPUT
	(* for the test it's the parameter ``lowerLimit`` *)
	lowerLimit	:REAL;
	(* for the test it's the parameter ``currentValue`` *)
	valueToTest	:REAL;
	(* for the test it's the parameter ``upperLimit`` *)
	upperLimit	:REAL;
END_VAR
VAR
	(* just the expectation if the assertion to test must be worng or true *)
	assertionIsWrong		:BOOL;
	(* contains the format string for the test message *)
	message					:Tc2_System.T_MaxString;
	(* TwinCAT printf with the test message *)
	messageStringBuilder	:Tc2_Utilities.FB_FormatString;
	(* just to cast *)
	binaryLowerLimit		:POINTER TO DWORD;
	(* just to cast *)
	binaryCurrentValue		:POINTER TO DWORD;
	(* just to cast *)
	binaryUpperLimit		:POINTER TO DWORD;
	(* value of the paramter ``lowerLimit`` as string *)
	lowerLimitAsString		:Tc2_System.T_MaxString;
	(* value of the paramter ``valueToTest`` as string *)
	valueToTestAsString		:Tc2_System.T_MaxString;
	(* value of the paramter ``upperLimit`` as string *)
	upperLimitAsString		:Tc2_System.T_MaxString;	
END_VAR
THIS^.assertorContainer.resetAssertor();

IF (
	Tc2_Utilities.RealIsNaN(lowerLimit)
	OR Tc2_Utilities.RealIsNaN(valueToTest)
	OR  Tc2_Utilities.RealIsNaN(upperLimit)
) THEN
	assertionIsWrong := TRUE;
ELSIF (
	(NOT Tc2_Utilities.RealIsFinite(lowerLimit))
	AND (NOT Tc2_Utilities.RealIsFinite(valueToTest))
	AND (NOT Tc2_Utilities.RealIsFinite(upperLimit))
) THEN
	binaryLowerLimit	:= ADR(lowerLimit);
	binaryCurrentValue	:= ADR(valueToTest);
	binaryUpperLimit	:= ADR(upperLimit);
	assertionIsWrong := (
		((NOT binaryLowerLimit^.SIGN) AND binaryUpperLimit^.SIGN)
		OR (
			((NOT binaryLowerLimit^.SIGN) AND (NOT binaryUpperLimit^.SIGN) AND binaryCurrentValue^.SIGN)
		) OR (
			(binaryLowerLimit^.SIGN AND binaryUpperLimit^.SIGN AND (NOT binaryCurrentValue^.SIGN))
		)
	);
ELSIF (
	(Tc2_Utilities.RealIsFinite(lowerLimit))
	AND (NOT Tc2_Utilities.RealIsFinite(valueToTest))
	AND (Tc2_Utilities.RealIsFinite(upperLimit))
) THEN
	assertionIsWrong := TRUE;
ELSIF (
	(NOT Tc2_Utilities.RealIsFinite(lowerLimit))
	AND (Tc2_Utilities.RealIsFinite(valueToTest))
	AND (Tc2_Utilities.RealIsFinite(upperLimit))
) THEN
	binaryLowerLimit	:= ADR(lowerLimit);
	assertionIsWrong := (
		(NOT binaryLowerLimit^.SIGN)
		OR (valueToTest > upperLimit)
	);
ELSIF (
	(Tc2_Utilities.RealIsFinite(lowerLimit))
	AND (Tc2_Utilities.RealIsFinite(valueToTest))
	AND (NOT Tc2_Utilities.RealIsFinite(upperLimit))
) THEN
	binaryUpperLimit	:= ADR(upperLimit);
	assertionIsWrong := (
		(binaryUpperLimit^.SIGN)
		OR (valueToTest < lowerLimit)
	);
ELSE
	assertionIsWrong := assertionIsWrong := ((valueToTest < lowerLimit) OR (valueToTest > upperLimit));
END_IF

message := SEL(
	assertionIsWrong,
	'lowerLimit is %s currentValue is %s upperLimit is %s assertion must be TRUE', 
	'lowerLimit is %s currentValue is %s upperLimit is %s assertion must be FALSE'
);

lowerLimitAsString	:= TO_STRING(lowerLimit);
valueToTestAsString := TO_STRING(valueToTest);
upperLimitAsString  := TO_STRING(upperLimit);

messageStringBuilder(
	sFormat := message,
	arg1 := THIS^.AnyToArg(lowerLimitAsString),
	arg2 := THIS^.AnyToArg(valueToTestAsString),
	arg3 := THIS^.AnyToArg(upperLimitAsString)
);

THIS^.assertorContainer.assertor.assert.float.single.valueIsInRangeOf(
	lowerLimit		:= lowerLimit,
	currentValue	:= valueToTest,
	upperLimit		:= upperLimit,
	message			:= ''
);

THIS^.AssertEquals_BOOL(
	Expected 	:= assertionIsWrong,
	Actual 		:= THIS^.assertorContainer.wasAssertionWrong,
	Message 	:= messageStringBuilder.sOut
);
END_METHOD

(*

short summary
==================
This test method tests ``assert.float.single.valueIsLessThan``
method of CNM_AssertionInterfaces library, 
it provides the possibility to handover test data via parameter 


.. <legal notes>

legal notes
=================
| SPDX-FileCopyrightText: © 2022 ekvip automation GmbH <info@ekvip.de>
| SPDX-License-Identifier: Apache-2.0
| For details check: Apache-2.0_

.. _Apache-2.0: https://www.apache.org/licenses/LICENSE-2.0

.. </legal notes>

parameters
==========

*)

METHOD testValueIsLessThan 
VAR_INPUT
	(* for the test it's the parameter ``currentValue`` *)
	valueToTest		:REAL;
	(* for the test it's the parameter ``greaterValue`` *)
	greaterValue	:REAL;
END_VAR
VAR
	(* just the expectation if the assertion to test must be worng or true *)
	assertionIsWrong		:BOOL;
	(* contains the format string for the test message *)
	message					:Tc2_System.T_MaxString;
	(* TwinCAT printf with the test message *)
	messageStringBuilder	:Tc2_Utilities.FB_FormatString;
	(* just to cast *)
	binaryCurrentValue		:POINTER TO DWORD;
	(* just to cast *)
	binaryGreaterValue		:POINTER TO DWORD;
	(* value of the paramter ``valueToTest`` as string *)
	valueToTestAsString		:Tc2_System.T_MaxString;
	(* value of the paramter ``greaterValue`` as string *)
	greaterValueAsString	:Tc2_System.T_MaxString;	
END_VAR
THIS^.assertorContainer.resetAssertor();

IF (Tc2_Utilities.RealIsNaN(valueToTest) OR Tc2_Utilities.RealIsNaN(greaterValue)) THEN
	assertionIsWrong := TRUE;
ELSIF ((NOT Tc2_Utilities.RealIsFinite(valueToTest)) AND (NOT Tc2_Utilities.RealIsFinite(greaterValue))) THEN
	binaryCurrentValue := ADR(valueToTest);
	binaryGreaterValue := ADR(greaterValue);
	assertionIsWrong := (
		(NOT binaryCurrentValue^.SIGN) //inf
		OR (binaryGreaterValue^.SIGN) //-inf
	);
ELSIF ((NOT Tc2_Utilities.RealIsFinite(valueToTest)) AND (Tc2_Utilities.RealIsFinite(greaterValue))) THEN
	binaryCurrentValue := ADR(valueToTest);
	assertionIsWrong := (NOT binaryCurrentValue^.SIGN); //inf
ELSIF ((Tc2_Utilities.RealIsFinite(valueToTest)) AND (NOT Tc2_Utilities.RealIsFinite(greaterValue))) THEN
	binaryGreaterValue := ADR(greaterValue);
	assertionIsWrong := (binaryGreaterValue^.SIGN); //-inf
ELSE
	assertionIsWrong := (valueToTest >= greaterValue);
END_IF

message := SEL(
	assertionIsWrong,
	'currentValue is %s greaterValue is %s assertion must be TRUE', 
	'currentValue is %s greaterValue is %s assertion must be FALSE'
);

valueToTestAsString := TO_STRING(valueToTest);
greaterValueAsString := TO_STRING(greaterValue);

messageStringBuilder(
	sFormat := message,
	arg1 := THIS^.AnyToArg(valueToTestAsString),
	arg2 := THIS^.AnyToArg(greaterValueAsString)
);

THIS^.assertorContainer.assertor.assert.float.single.valueIsLessThan(
	currentValue	:= valueToTest,
	greaterValue	:= greaterValue,
	message			:= ''
);

THIS^.AssertEquals_BOOL(
	Expected 	:= assertionIsWrong,
	Actual 		:= THIS^.assertorContainer.wasAssertionWrong,
	Message 	:= messageStringBuilder.sOut
);
END_METHOD

(*

short summary
==================
This test method tests ``assert.float.single.valueIsMax``
method of CNM_AssertionInterfaces library, 
it provides the possibility to handover test data via parameter 


.. <legal notes>

legal notes
=================
| SPDX-FileCopyrightText: © 2022 ekvip automation GmbH <info@ekvip.de>
| SPDX-License-Identifier: Apache-2.0
| For details check: Apache-2.0_

.. _Apache-2.0: https://www.apache.org/licenses/LICENSE-2.0

.. </legal notes>

parameters
==========

*)

METHOD testValueIsMax 
VAR_INPUT
	(* for the test it's the parameter ``currentValue`` *)
	valueToTest		:REAL;
	(* for the test it's the parameter ``greaterValue`` *)
	maximumValue	:REAL;
END_VAR
VAR
	(* just the expectation if the assertion to test must be worng or true *)
	assertionIsWrong		:BOOL;
	(* contains the format string for the test message *)
	message					:Tc2_System.T_MaxString;
	(* TwinCAT printf with the test message *)
	messageStringBuilder	:Tc2_Utilities.FB_FormatString;
	(* just to cast *)
	binaryCurrentValue		:POINTER TO DWORD;
	(* just to cast *)
	binaryMaximumValue		:POINTER TO DWORD;
	(* value of the paramter ``valueToTest`` as string *)
	valueToTestAsString		:Tc2_System.T_MaxString;
	(* value of the paramter ``maximumValue`` as string *)
	maximumValueAsString	:Tc2_System.T_MaxString;	
END_VAR
THIS^.assertorContainer.resetAssertor();

IF (Tc2_Utilities.RealIsNaN(valueToTest) OR Tc2_Utilities.RealIsNaN(maximumValue)) THEN
	assertionIsWrong := TRUE;
ELSIF ((NOT Tc2_Utilities.RealIsFinite(valueToTest)) AND (NOT Tc2_Utilities.RealIsFinite(maximumValue))) THEN
	binaryCurrentValue := ADR(valueToTest);
	binaryMaximumValue := ADR(maximumValue);
	assertionIsWrong := (
		(NOT binaryCurrentValue^.SIGN) //inf
		AND (binaryMaximumValue^.SIGN) //-inf
	);
ELSIF ((NOT Tc2_Utilities.RealIsFinite(valueToTest)) AND (Tc2_Utilities.RealIsFinite(maximumValue))) THEN
	binaryCurrentValue := ADR(valueToTest);
	assertionIsWrong := (NOT binaryCurrentValue^.SIGN); //inf
ELSIF ((Tc2_Utilities.RealIsFinite(valueToTest)) AND (NOT Tc2_Utilities.RealIsFinite(maximumValue))) THEN
	binaryMaximumValue := ADR(maximumValue);
	assertionIsWrong := (binaryMaximumValue^.SIGN);//-inf
ELSE
	assertionIsWrong := (valueToTest > maximumValue);
END_IF

message := SEL(
	assertionIsWrong,
	'currentValue is %s maximumValue is %s assertion must be TRUE', 
	'currentValue is %s maximumValue is %s assertion must be FALSE'
);

valueToTestAsString := TO_STRING(valueToTest);
maximumValueAsString := TO_STRING(maximumValue);

messageStringBuilder(
	sFormat := message,
	arg1 := THIS^.AnyToArg(valueToTestAsString),
	arg2 := THIS^.AnyToArg(maximumValueAsString)
);

THIS^.assertorContainer.assertor.assert.float.single.valueIsMax(
	currentValue	:= valueToTest,
	maximumValue	:= maximumValue,
	message			:= ''
);

THIS^.AssertEquals_BOOL(
	Expected 	:= assertionIsWrong,
	Actual 		:= THIS^.assertorContainer.wasAssertionWrong,
	Message 	:= messageStringBuilder.sOut
);
END_METHOD

(*

short summary
==================
This test method tests ``assert.float.single.valueIsMin``
method of CNM_AssertionInterfaces library, 
it provides the possibility to handover test data via parameter 


.. <legal notes>

legal notes
=================
| SPDX-FileCopyrightText: © 2022 ekvip automation GmbH <info@ekvip.de>
| SPDX-License-Identifier: Apache-2.0
| For details check: Apache-2.0_

.. _Apache-2.0: https://www.apache.org/licenses/LICENSE-2.0

.. </legal notes>

parameters
==========

*)

METHOD testValueIsMin 
VAR_INPUT
	(* for the test it's the parameter ``currentValue`` *)
	valueToTest		:REAL;
	(* for the test it's the parameter ``greaterValue`` *)
	minimumValue	:REAL;
END_VAR
VAR
	(* just the expectation if the assertion to test must be worng or true *)
	assertionIsWrong		:BOOL;
	(* contains the format string for the test message *)
	message					:Tc2_System.T_MaxString;
	(* TwinCAT printf with the test message *)
	messageStringBuilder	:Tc2_Utilities.FB_FormatString;
	(* just to cast *)
	binaryCurrentValue		:POINTER TO DWORD;
	(* just to cast *)
	binaryMinimumValue		:POINTER TO DWORD;
	(* value of the paramter ``valueToTest`` as string *)
	valueToTestAsString		:Tc2_System.T_MaxString;
	(* value of the paramter ``minimumValue`` as string *)
	minimumValueAsString	:Tc2_System.T_MaxString;	
END_VAR
THIS^.assertorContainer.resetAssertor();

IF (Tc2_Utilities.RealIsNaN(valueToTest) OR Tc2_Utilities.RealIsNaN(minimumValue)) THEN
	assertionIsWrong := TRUE;
ELSIF ((NOT Tc2_Utilities.RealIsFinite(valueToTest)) AND (NOT Tc2_Utilities.RealIsFinite(minimumValue))) THEN
	binaryCurrentValue := ADR(valueToTest);
	binaryMinimumValue := ADR(minimumValue);
	assertionIsWrong := (
		(binaryCurrentValue^.SIGN) //-inf
		AND (NOT binaryMinimumValue^.SIGN) //inf
	);
ELSIF ((NOT Tc2_Utilities.RealIsFinite(valueToTest)) AND (Tc2_Utilities.RealIsFinite(minimumValue))) THEN
	binaryCurrentValue := ADR(valueToTest);
	assertionIsWrong := (binaryCurrentValue^.SIGN);
ELSIF ((Tc2_Utilities.RealIsFinite(valueToTest)) AND (NOT Tc2_Utilities.RealIsFinite(minimumValue))) THEN
	binaryMinimumValue := ADR(minimumValue);
	assertionIsWrong := (NOT binaryMinimumValue^.SIGN);
ELSE
	assertionIsWrong := (valueToTest < minimumValue);
END_IF

message := SEL(
	assertionIsWrong,
	'currentValue is %s minimumValue is %s assertion must be TRUE', 
	'currentValue is %s minimumValue is %s assertion must be FALSE'
);

valueToTestAsString := TO_STRING(valueToTest);
minimumValueAsString := TO_STRING(minimumValue);

messageStringBuilder(
	sFormat := message,
	arg1 := THIS^.AnyToArg(valueToTestAsString),
	arg2 := THIS^.AnyToArg(minimumValueAsString)
);

THIS^.assertorContainer.assertor.assert.float.single.valueIsMin(
	currentValue	:= valueToTest,
	minimumValue	:= minimumValue,
	message			:= ''
);

THIS^.AssertEquals_BOOL(
	Expected 	:= assertionIsWrong,
	Actual 		:= THIS^.assertorContainer.wasAssertionWrong,
	Message 	:= messageStringBuilder.sOut
);
END_METHOD

(*

short summary
==================
This test method tests ``assert.float.single.valueIsNaN``
method of CNM_AssertionInterfaces library, 
it provides the possibility to handover test data via parameter 

.. <legal notes>

legal notes
=================
| SPDX-FileCopyrightText: © 2022 ekvip automation GmbH <info@ekvip.de>
| SPDX-License-Identifier: Apache-2.0
| For details check: Apache-2.0_

.. _Apache-2.0: https://www.apache.org/licenses/LICENSE-2.0

.. </legal notes>

parameters
==========

*)

METHOD testValueIsNaN
VAR_INPUT
	(* for the test it's the parameter ``currentValue`` *)
	valueToTest	:REAL;	
END_VAR
VAR
	(* just the expectation if the assertion to test must be worng or true *)
	assertionIsWrong		:BOOL;
	(* contains the format string for the test message *)
	message					:Tc2_System.T_MaxString;
	(* TwinCAT printf with the test message *)
	messageStringBuilder	:Tc2_Utilities.FB_FormatString;
	(* value of the paramter ``valueToTest`` as string *)
	valueToTestAsString		:Tc2_System.T_MaxString;
END_VAR
THIS^.assertorContainer.resetAssertor();

assertionIsWrong := (NOT Tc2_Utilities.RealIsNaN(valueToTest));

message := SEL(
	assertionIsWrong,
	'currentValue is %s assertion must be TRUE', 
	'currentValue is %s assertion must be FALSE'
);

valueToTestAsString := TO_STRING(valueToTest);

messageStringBuilder(
	sFormat := message,
	arg1 := THIS^.AnyToArg(valueToTestAsString)
);

THIS^.assertorContainer.assertor.assert.float.single.valueIsNaN(
	currentValue := valueToTest,
	message := ''
);

THIS^.AssertEquals_BOOL(
	Expected 	:= assertionIsWrong,
	Actual 		:= THIS^.assertorContainer.wasAssertionWrong,
	Message 	:= messageStringBuilder.sOut
);
END_METHOD

(*

short summary
==================
This test method tests ``assert.float.single.valueIsNegative``
method of CNM_AssertionInterfaces library, 
it provides the possibility to handover test data via parameter 

.. <legal notes>

legal notes
=================
| SPDX-FileCopyrightText: © 2022 ekvip automation GmbH <info@ekvip.de>
| SPDX-License-Identifier: Apache-2.0
| For details check: Apache-2.0_

.. _Apache-2.0: https://www.apache.org/licenses/LICENSE-2.0

.. </legal notes>

parameters
==========

*)

METHOD testValueIsNegative
VAR_INPUT
	(* for the test it's the parameter ``currentValue`` *)
	valueToTest	:REAL;	
END_VAR
VAR
	(* just the expectation if the assertion to test must be worng or true *)
	assertionIsWrong		:BOOL;
	(* contains the format string for the test message *)
	message					:Tc2_System.T_MaxString;
	(* TwinCAT printf with the test message *)
	messageStringBuilder	:Tc2_Utilities.FB_FormatString;
	(* value of the paramter ``valueToTest`` as string *)
	valueToTestAsString		:Tc2_System.T_MaxString;
	(* binary value of the parameter ``valueToTest`` *)
	binaryValueToTest		:POINTER TO DWORD;
	(* sgin bit as BYTE for the message *)
	signBitAsByte			:BYTE;
	(* sgin bit as BOOL for the message *)
	signBit					:BOOL;	
END_VAR
THIS^.assertorContainer.resetAssertor();

binaryValueToTest := ADR(valueToTest);
signBit := binaryValueToTest^.SIGN;
signBitAsByte := TO_BYTE(signBit);
assertionIsWrong := (
	(NOT signBit)
	OR_ELSE Tc2_Utilities.RealIsNaN(valueToTest)
);

message := SEL(
	assertionIsWrong,
	'currentValue is %s and sign bit is %u assertion must be TRUE', 
	'currentValue is %s and sign bit is %u assertion must be FALSE'
);

valueToTestAsString := TO_STRING(valueToTest);

messageStringBuilder(
	sFormat := message,
	arg1 := THIS^.AnyToArg(valueToTestAsString),
	arg2 := THIS^.AnyToArg(signBitAsByte)
);

THIS^.assertorContainer.assertor.assert.float.single.valueIsNegative(
	currentValue := valueToTest,
	message := ''
);

THIS^.AssertEquals_BOOL(
	Expected 	:= assertionIsWrong,
	Actual 		:= THIS^.assertorContainer.wasAssertionWrong,
	Message 	:= messageStringBuilder.sOut
);
END_METHOD

(*

short summary
==================
This test method tests ``assert.float.single.valueIsNegativeInfinite``
method of CNM_AssertionInterfaces library, 
it provides the possibility to handover test data via parameter 

.. <legal notes>

legal notes
=================
| SPDX-FileCopyrightText: © 2022 ekvip automation GmbH <info@ekvip.de>
| SPDX-License-Identifier: Apache-2.0
| For details check: Apache-2.0_

.. _Apache-2.0: https://www.apache.org/licenses/LICENSE-2.0

.. </legal notes>

parameters
==========

*)

METHOD testValueIsNegativeInfinite
VAR_INPUT
	(* for the test it's the parameter ``currentValue`` *)
	valueToTest	:REAL;	
END_VAR
VAR
	(* just the expectation if the assertion to test must be worng or true *)
	assertionIsWrong		:BOOL;
	(* contains the format string for the test message *)
	message					:Tc2_System.T_MaxString;
	(* TwinCAT printf with the test message *)
	messageStringBuilder	:Tc2_Utilities.FB_FormatString;
	(* value of the paramter ``valueToTest`` as string *)
	valueToTestAsString		:Tc2_System.T_MaxString;
	(* binary value of the parameter ``valueToTest`` *)
	binaryValueToTest		:POINTER TO DWORD;
END_VAR
THIS^.assertorContainer.resetAssertor();

